C09132=1229.334,-18.388,-40.165,-179.651,5.314,148.817
C09133=1229.329,-18.138,-40.179,-179.649,5.313,148.816
C09134=1229.323,-17.889,-40.193,-179.646,5.314,148.816
C09135=1229.319,-17.639,-40.206,-179.643,5.314,148.815
C09136=1229.314,-17.390,-40.221,-179.641,5.314,148.814
C09137=1229.308,-17.141,-40.235,-179.638,5.315,148.813
C09138=1229.303,-16.890,-40.248,-179.636,5.315,148.813
C09139=1229.299,-16.641,-40.262,-179.634,5.315,148.812
C09140=1229.293,-16.392,-40.276,-179.631,5.315,148.811
C09141=1229.288,-16.142,-40.289,-179.628,5.316,148.810
C09142=1229.283,-15.892,-40.304,-179.626,5.315,148.810
C09143=1229.278,-15.643,-40.317,-179.623,5.316,148.809
C09144=1229.273,-15.394,-40.331,-179.621,5.316,148.808
C09145=1229.268,-15.143,-40.345,-179.618,5.316,148.808
C09146=1229.262,-14.894,-40.359,-179.616,5.316,148.807
C09147=1229.258,-14.645,-40.372,-179.613,5.317,148.806
C09148=1229.253,-14.395,-40.387,-179.611,5.317,148.806
C09149=1229.247,-14.145,-40.400,-179.608,5.317,148.805
C09150=1229.242,-13.896,-40.414,-179.606,5.318,148.804
C09151=1229.237,-13.646,-40.428,-179.604,5.317,148.803
C09152=1229.233,-13.397,-40.442,-179.601,5.318,148.803
C09153=1229.228,-13.148,-40.456,-179.598,5.318,148.802
C09154=1229.222,-12.897,-40.469,-179.596,5.319,148.801
C09155=1229.217,-12.648,-40.483,-179.594,5.319,148.801
C09156=1229.212,-12.399,-40.498,-179.591,5.319,148.800
C09157=1229.208,-12.149,-40.511,-179.588,5.320,148.799
C09158=1229.203,-11.899,-40.526,-179.586,5.319,148.799
C09159=1229.197,-11.650,-40.540,-179.584,5.320,148.798
C09160=1229.192,-11.400,-40.553,-179.581,5.320,148.797
C09161=1229.187,-11.150,-40.567,-179.579,5.320,148.797
C09162=1229.182,-10.901,-40.582,-179.576,5.321,148.796
C09163=1229.176,-10.652,-40.596,-179.573,5.321,148.795
C09164=1229.172,-10.402,-40.609,-179.571,5.321,148.794
C09165=1229.167,-10.153,-40.624,-179.569,5.321,148.794
C09166=1229.162,-9.904,-40.637,-179.566,5.322,148.793
C09167=1229.157,-9.654,-40.652,-179.564,5.322,148.792
C09168=1229.152,-9.404,-40.666,-179.561,5.322,148.792
C09169=1229.147,-9.154,-40.680,-179.559,5.323,148.791
C09170=1229.142,-8.904,-40.694,-179.556,5.323,148.790
C09171=1229.136,-8.655,-40.708,-179.554,5.323,148.790
C09172=1229.131,-8.405,-40.722,-179.551,5.323,148.789
C09173=1229.127,-8.156,-40.736,-179.549,5.324,148.788
C09174=1229.122,-7.906,-40.750,-179.547,5.324,148.788
C09175=1229.116,-7.657,-40.764,-179.544,5.324,148.787
C09176=1229.111,-7.408,-40.778,-179.541,5.325,148.786
C09177=1229.106,-7.158,-40.792,-179.539,5.324,148.785
C09178=1229.102,-6.908,-40.807,-179.537,5.325,148.785
C09179=1229.097,-6.658,-40.821,-179.534,5.325,148.784
C09180=1229.091,-6.409,-40.835,-179.531,5.326,148.783
C09181=1229.086,-6.160,-40.849,-179.529,5.326,148.783
C09182=1229.081,-5.910,-40.863,-179.527,5.326,148.782
C09183=1229.076,-5.660,-40.878,-179.524,5.327,148.781
C09184=1229.071,-5.411,-40.892,-179.522,5.326,148.781
C09185=1229.066,-5.162,-40.906,-179.519,5.327,148.780
C09186=1229.061,-4.912,-40.920,-179.516,5.327,148.779
C09187=1229.056,-4.663,-40.935,-179.514,5.327,148.779
C09188=1229.051,-4.413,-40.949,-179.512,5.328,148.778
C09189=1229.046,-4.163,-40.964,-179.509,5.328,148.777
C09190=1229.041,-3.914,-40.978,-179.506,5.329,148.777
C09191=1229.036,-3.665,-40.992,-179.504,5.328,148.776
C09192=1229.031,-3.415,-41.006,-179.502,5.329,148.775
C09193=1229.026,-3.165,-41.021,-179.499,5.329,148.774
C09194=1229.021,-2.915,-41.035,-179.497,5.329,148.774
C09195=1229.016,-2.666,-41.049,-179.494,5.330,148.773
C09196=1229.011,-2.416,-41.063,-179.492,5.330,148.772
C09197=1229.006,-2.168,-41.078,-179.489,5.331,148.772
C09198=1229.001,-1.918,-41.092,-179.487,5.330,148.771
C09199=1228.996,-1.668,-41.107,-179.484,5.331,148.770
C09200=1228.991,-1.419,-41.121,-179.482,5.331,148.770
C09201=1228.986,-1.169,-41.135,-179.480,5.331,148.769
C09202=1228.981,-0.919,-41.149,-179.477,5.332,148.768
C09203=1228.976,-0.670,-41.164,-179.474,5.332,148.768
C09204=1228.970,-0.420,-41.179,-179.472,5.333,148.767
C09205=1228.965,-0.171,-41.193,-179.469,5.332,148.766
C09206=1228.960,0.079,-41.207,-179.467,5.333,148.765
C09207=1228.955,0.328,-41.222,-179.464,5.334,148.765
C09208=1228.950,0.578,-41.237,-179.462,5.334,148.764
C09209=1228.945,0.827,-41.251,-179.459,5.334,148.763
C09210=1228.940,1.077,-41.265,-179.456,5.334,148.762
C09211=1228.936,1.327,-41.280,-179.454,5.334,148.762
C09212=1228.931,1.576,-41.294,-179.452,5.334,148.761
C09213=1228.925,1.826,-41.309,-179.449,5.335,148.760
C09214=1228.920,2.075,-41.324,-179.446,5.335,148.760
C09215=1228.915,2.324,-41.338,-179.444,5.336,148.759
C09216=1228.910,2.574,-41.353,-179.442,5.335,148.758
C09217=1228.905,2.823,-41.367,-179.439,5.336,148.758
C09218=1228.900,3.073,-41.381,-179.436,5.337,148.757
C09219=1228.894,3.342,-41.397,-179.434,5.337,148.756
C09220=1228.889,3.611,-41.413,-179.431,5.338,148.756
C09221=1228.884,3.880,-41.429,-179.429,5.337,148.755
C09222=1228.879,4.148,-41.445,-179.426,5.338,148.754
C09223=1228.873,4.399,-41.459,-179.424,5.338,148.754
C09224=1228.868,4.648,-41.474,-179.421,5.339,148.753
C09225=1228.864,4.897,-41.489,-179.418,5.339,148.752
C09226=1228.859,5.147,-41.503,-179.416,5.339,148.751
C09227=1228.854,5.396,-41.518,-179.414,5.340,148.751
C09228=1228.848,5.646,-41.533,-179.411,5.340,148.750
C09229=1228.843,5.896,-41.547,-179.408,5.341,148.749
C09230=1228.839,6.145,-41.562,-179.406,5.340,148.749
C09231=1228.834,6.395,-41.576,-179.403,5.341,148.748
C09232=1228.828,6.644,-41.592,-179.401,5.342,148.747
C09233=1228.823,6.894,-41.606,-179.398,5.342,148.747
C09234=1228.818,7.143,-41.621,-179.396,5.342,148.746
C09235=1228.814,7.393,-41.635,-179.393,5.342,148.745
C09236=1228.808,7.643,-41.650,-179.391,5.343,148.745
C09237=1228.803,7.892,-41.665,-179.388,5.343,148.744
C09238=1228.798,8.141,-41.680,-179.386,5.343,148.743
C09239=1228.794,8.390,-41.695,-179.383,5.344,148.743
C09240=1228.788,8.641,-41.710,-179.381,5.344,148.742
C09241=1228.783,8.890,-41.724,-179.378,5.345,148.741
C09242=1228.779,9.139,-41.739,-179.376,5.344,148.740
C09243=1228.773,9.389,-41.754,-179.373,5.345,148.740
C09244=1228.768,9.638,-41.769,-179.371,5.345,148.739
C09245=1228.764,9.888,-41.784,-179.368,5.346,148.738
C09246=1228.759,10.137,-41.798,-179.366,5.346,148.738
C09247=1228.753,10.387,-41.813,-179.363,5.346,148.737
C09248=1228.748,10.636,-41.828,-179.361,5.347,148.736
C09249=1228.744,10.885,-41.843,-179.358,5.347,148.736
C09250=1228.738,11.135,-41.858,-179.356,5.347,148.735
C09251=1228.733,11.385,-41.873,-179.353,5.348,148.734
C09252=1228.728,11.634,-41.888,-179.351,5.348,148.734
C09253=1228.723,11.884,-41.902,-179.348,5.349,148.733
C09254=1228.718,12.133,-41.917,-179.346,5.348,148.732
C09255=1228.713,12.383,-41.932,-179.343,5.349,148.732
C09256=1228.708,12.632,-41.947,-179.341,5.349,148.731
C09257=1228.703,12.882,-41.962,-179.338,5.350,148.730
C09258=1228.698,13.131,-41.977,-179.335,5.351,148.730
C09259=1228.693,13.380,-41.992,-179.333,5.350,148.729
C09260=1228.688,13.631,-42.007,-179.331,5.351,148.728
C09261=1228.683,13.880,-42.022,-179.328,5.351,148.727
C09262=1228.679,14.129,-42.037,-179.325,5.352,148.727
C09263=1228.673,14.379,-42.052,-179.323,5.352,148.726
C09264=1228.668,14.628,-42.067,-179.321,5.352,148.725
C09265=1228.663,14.877,-42.083,-179.318,5.353,148.725
C09266=1228.658,15.127,-42.097,-179.315,5.353,148.724
C09267=1228.653,15.376,-42.112,-179.313,5.354,148.723
C09268=1228.648,15.626,-42.128,-179.311,5.353,148.723
C09269=1228.643,15.875,-42.142,-179.308,5.354,148.722
C09270=1228.638,16.125,-42.158,-179.305,5.355,148.721
C09271=1228.633,16.375,-42.173,-179.303,5.355,148.721
C09272=1228.628,16.624,-42.189,-179.301,5.355,148.720
C09273=1228.623,16.874,-42.203,-179.298,5.355,148.719
C09274=1228.618,17.123,-42.218,-179.295,5.356,148.719
C09275=1228.613,17.372,-42.233,-179.293,5.356,148.718
C09276=1228.608,17.622,-42.249,-179.290,5.357,148.717
C09277=1228.603,17.872,-42.264,-179.288,5.357,148.717
C09278=1228.598,18.121,-42.279,-179.285,5.357,148.716
C09279=1228.593,18.370,-42.294,-179.283,5.358,148.715
C09280=1228.588,18.620,-42.310,-179.280,5.359,148.715
C09281=1228.583,18.869,-42.325,-179.278,5.359,148.714
C09282=1228.578,19.119,-42.340,-179.276,5.359,148.713
C09283=1228.573,19.368,-42.355,-179.273,5.359,148.713
C09284=1228.568,19.618,-42.371,-179.270,5.360,148.712
C09285=1228.563,19.867,-42.386,-179.268,5.361,148.711
C09286=1228.558,20.117,-42.401,-179.265,5.361,148.711
C09287=1228.553,20.366,-42.416,-179.263,5.361,148.710
C09288=1228.548,20.616,-42.431,-179.260,5.361,148.709
C09289=1228.544,20.866,-42.446,-179.258,5.362,148.709
C09290=1228.538,21.115,-42.462,-179.255,5.362,148.708
C09291=1228.533,21.364,-42.478,-179.253,5.363,148.707
C09292=1228.528,21.613,-42.493,-179.250,5.363,148.707
C09293=1228.523,21.863,-42.508,-179.248,5.363,148.706
C09294=1228.519,22.113,-42.524,-179.245,5.364,148.705
C09295=1228.513,22.362,-42.539,-179.243,5.364,148.704
C09296=1228.508,22.612,-42.554,-179.240,5.365,148.704
C09297=1228.503,22.861,-42.569,-179.238,5.365,148.703
C09298=1228.498,23.111,-42.585,-179.235,5.365,148.702
C09299=1228.494,23.360,-42.600,-179.232,5.366,148.702
C09300=1228.488,23.610,-42.616,-179.230,5.366,148.701
C09301=1228.483,23.859,-42.631,-179.227,5.367,148.700
C09302=1228.478,24.108,-42.646,-179.225,5.367,148.700
C09303=1228.473,24.358,-42.662,-179.222,5.367,148.699
C09304=1228.468,24.608,-42.678,-179.220,5.368,148.698
C09305=1228.463,24.857,-42.693,-179.217,5.368,148.698
C09306=1228.458,25.106,-42.708,-179.215,5.369,148.697
C09307=1228.454,25.356,-42.724,-179.212,5.370,148.697
C09308=1228.449,25.605,-42.739,-179.210,5.369,148.696
C09309=1228.443,25.855,-42.755,-179.208,5.370,148.695
C09310=1228.439,26.104,-42.770,-179.205,5.370,148.694
C09311=1228.434,26.354,-42.786,-179.202,5.371,148.694
C09312=1228.428,26.603,-42.801,-179.200,5.372,148.693
C09313=1228.423,26.853,-42.817,-179.197,5.372,148.692
C09314=1228.418,27.102,-42.832,-179.195,5.372,148.692
C09315=1228.414,27.351,-42.849,-179.192,5.372,148.691
C09316=1228.408,27.601,-42.864,-179.190,5.373,148.690
C09317=1228.404,27.850,-42.879,-179.187,5.373,148.690
C09318=1228.399,28.100,-42.895,-179.184,5.374,148.689
C09319=1228.394,28.349,-42.911,-179.182,5.375,148.688
C09320=1228.388,28.599,-42.926,-179.180,5.374,148.688
C09321=1228.384,28.849,-42.942,-179.177,5.375,148.687
C09322=1228.379,29.098,-42.957,-179.174,5.375,148.686
C09323=1228.373,29.367,-42.974,-179.172,5.376,148.686
C09324=1228.368,29.635,-42.991,-179.169,5.377,148.685
C09325=1228.363,29.903,-43.008,-179.167,5.377,148.684
C09326=1228.358,30.172,-43.025,-179.164,5.378,148.684
C09327=1228.353,30.422,-43.041,-179.161,5.378,148.683
C09328=1228.347,30.671,-43.056,-179.159,5.379,148.682
C09329=1228.342,30.921,-43.072,-179.156,5.379,148.682
C09330=1228.338,31.170,-43.087,-179.154,5.379,148.681
C09331=1228.333,31.419,-43.103,-179.151,5.380,148.680
C09332=1228.328,31.669,-43.119,-179.149,5.380,148.680
C09333=1228.322,31.919,-43.135,-179.146,5.381,148.679
C09334=1228.317,32.168,-43.151,-179.143,5.381,148.678
C09335=1228.313,32.417,-43.167,-179.141,5.382,148.678
C09336=1228.308,32.667,-43.182,-179.139,5.382,148.677
C09337=1228.303,32.916,-43.198,-179.136,5.382,148.676
C09338=1228.298,33.166,-43.214,-179.133,5.383,148.675
C09339=1228.293,33.415,-43.230,-179.131,5.383,148.675
C09340=1228.287,33.664,-43.246,-179.129,5.384,148.674
C09341=1228.283,33.914,-43.261,-179.126,5.385,148.674
C09342=1228.278,34.164,-43.277,-179.123,5.385,148.673
C09343=1228.273,34.413,-43.293,-179.121,5.385,148.672
C09344=1228.268,34.662,-43.309,-179.119,5.385,148.672
C09345=1228.263,34.912,-43.324,-179.116,5.386,148.671
C09346=1228.258,35.161,-43.341,-179.113,5.387,148.670
C09347=1228.253,35.411,-43.357,-179.111,5.387,148.670
C09348=1228.248,35.661,-43.373,-179.108,5.388,148.669
C09349=1228.244,35.909,-43.388,-179.105,5.388,148.668
C09350=1228.238,36.159,-43.404,-179.103,5.388,148.668
C09351=1228.233,36.409,-43.420,-179.101,5.389,148.667
C09352=1228.228,36.658,-43.436,-179.098,5.389,148.666
C09353=1228.224,36.908,-43.452,-179.096,5.390,148.666
C09354=1228.219,37.156,-43.469,-179.093,5.391,148.665
C09355=1228.214,37.407,-43.484,-179.091,5.391,148.664
C09356=1228.208,37.656,-43.500,-179.088,5.392,148.664
C09357=1228.203,37.905,-43.516,-179.085,5.392,148.663
C09358=1228.198,38.155,-43.532,-179.083,5.392,148.662
C09359=1228.193,38.404,-43.549,-179.081,5.393,148.662
C09360=1228.189,38.654,-43.565,-179.078,5.393,148.661
C09361=1228.184,38.903,-43.581,-179.075,5.394,148.660
C09362=1228.179,39.153,-43.597,-179.073,5.394,148.660
C09363=1228.173,39.402,-43.612,-179.070,5.395,148.659
C09364=1228.169,39.652,-43.629,-179.067,5.395,148.658
C09365=1228.163,39.901,-43.645,-179.065,5.396,148.658
C09366=1228.159,40.150,-43.661,-179.063,5.396,148.657
C09367=1228.154,40.400,-43.677,-179.060,5.397,148.657
C09368=1228.149,40.649,-43.694,-179.058,5.397,148.656
C09369=1228.144,40.899,-43.709,-179.055,5.398,148.655
C09370=1228.139,41.147,-43.725,-179.053,5.398,148.655
C09371=1228.134,41.398,-43.741,-179.050,5.399,148.654
C09372=1228.129,41.646,-43.758,-179.047,5.399,148.653
C09373=1228.124,41.896,-43.774,-179.045,5.400,148.653
C09374=1228.119,42.145,-43.790,-179.042,5.401,148.652
C09375=1228.114,42.395,-43.807,-179.040,5.400,148.651
C09376=1228.109,42.644,-43.822,-179.038,5.401,148.651
C09377=1228.105,42.894,-43.839,-179.035,5.402,148.650
C09378=1228.100,43.144,-43.855,-179.032,5.402,148.649
C09379=1228.095,43.392,-43.871,-179.030,5.403,148.649
C09380=1228.090,43.642,-43.888,-179.027,5.403,148.648
C09381=1228.085,43.891,-43.903,-179.025,5.404,148.647
C09382=1228.080,44.141,-43.920,-179.022,5.405,148.647
C09383=1228.074,44.391,-43.936,-179.019,5.405,148.646
C09384=1228.070,44.640,-43.953,-179.017,5.406,148.645
C09385=1228.065,44.889,-43.969,-179.015,5.405,148.645
C09386=1228.060,45.139,-43.985,-179.012,5.406,148.644
C09387=1228.055,45.388,-44.002,-179.010,5.407,148.644
C09388=1228.050,45.637,-44.018,-179.007,5.407,148.643
C09389=1228.045,45.887,-44.034,-179.005,5.408,148.642
C09390=1228.040,46.136,-44.050,-179.002,5.409,148.642
C09391=1228.035,46.386,-44.068,-178.999,5.409,148.641
C09392=1228.030,46.635,-44.083,-178.997,5.410,148.640
C09393=1228.025,46.885,-44.100,-178.994,5.410,148.640
C09394=1228.020,47.134,-44.116,-178.991,5.411,148.639
C09395=1228.016,47.383,-44.133,-178.989,5.411,148.638
C09396=1228.010,47.632,-44.149,-178.987,5.412,148.638
C09397=1228.006,47.882,-44.165,-178.984,5.412,148.637
C09398=1228.001,48.132,-44.182,-178.982,5.413,148.636
C09399=1227.996,48.381,-44.199,-178.979,5.413,148.636
C09400=1227.991,48.631,-44.215,-178.977,5.414,148.635
C09401=1227.986,48.879,-44.231,-178.974,5.414,148.634
C09402=1227.981,49.129,-44.248,-178.971,5.415,148.634
C09403=1227.976,49.379,-44.265,-178.969,5.416,148.633
C09404=1227.971,49.627,-44.281,-178.967,5.416,148.633
C09405=1227.966,49.878,-44.297,-178.964,5.417,148.632
C09406=1227.962,50.127,-44.314,-178.961,5.418,148.631
C09407=1227.956,50.376,-44.331,-178.959,5.418,148.631
C09408=1227.951,50.626,-44.347,-178.956,5.419,148.630
C09409=1227.946,50.874,-44.364,-178.954,5.418,148.629
C09410=1227.942,51.124,-44.380,-178.951,5.419,148.629
C09411=1227.936,51.374,-44.397,-178.949,5.420,148.628
C09412=1227.931,51.623,-44.413,-178.946,5.420,148.627
C09413=1227.927,51.873,-44.430,-178.944,5.421,148.627
C09414=1227.922,52.122,-44.447,-178.941,5.422,148.626
C09415=1227.917,52.371,-44.464,-178.939,5.422,148.625
C09416=1227.912,52.621,-44.480,-178.936,5.423,148.625
C09417=1227.908,52.870,-44.497,-178.933,5.423,148.624
C09418=1227.902,53.119,-44.513,-178.931,5.424,148.623
C09419=1227.897,53.369,-44.530,-178.928,5.425,148.623
C09420=1227.892,53.619,-44.546,-178.926,5.425,148.622
C09421=1227.887,53.868,-44.563,-178.923,5.426,148.622
C09422=1227.882,54.117,-44.580,-178.921,5.427,148.621
C09423=1227.878,54.367,-44.597,-178.918,5.427,148.620
C09424=1227.873,54.616,-44.613,-178.915,5.428,148.620
C09425=1227.867,54.865,-44.630,-178.913,5.428,148.619
C09426=1227.863,55.115,-44.647,-178.911,5.428,148.618
C09427=1227.858,55.383,-44.665,-178.907,5.429,148.618
C09428=1227.852,55.652,-44.683,-178.905,5.430,148.617
C09429=1227.847,55.920,-44.701,-178.902,5.431,148.616
C09430=1227.842,56.188,-44.720,-178.900,5.431,148.616
C09431=1227.837,56.438,-44.736,-178.897,5.432,148.615
C09432=1227.832,56.687,-44.753,-178.894,5.432,148.614
C09433=1227.827,56.936,-44.770,-178.892,5.433,148.614
C09434=1227.822,57.186,-44.787,-178.889,5.434,148.613
C09435=1227.817,57.436,-44.804,-178.887,5.434,148.613
C09436=1227.812,57.685,-44.820,-178.884,5.435,148.612
C09437=1227.808,57.934,-44.837,-178.882,5.436,148.611
C09438=1227.802,58.184,-44.854,-178.879,5.436,148.611
C09439=1227.798,58.433,-44.871,-178.876,5.437,148.610
C09440=1227.792,58.682,-44.888,-178.874,5.436,148.609
C09441=1227.788,58.932,-44.904,-178.872,5.437,148.609
C09442=1227.783,59.181,-44.922,-178.869,5.438,148.608
C09443=1227.778,59.431,-44.939,-178.867,5.439,148.607
C09444=1227.772,59.680,-44.956,-178.864,5.439,148.607
C09445=1227.768,59.929,-44.973,-178.862,5.440,148.606
C09446=1227.763,60.179,-44.989,-178.859,5.440,148.605
C09447=1227.758,60.428,-45.006,-178.857,5.441,148.605
C09448=1227.753,60.677,-45.023,-178.854,5.442,148.604
C09449=1227.748,60.926,-45.041,-178.852,5.442,148.604
C09450=1227.744,61.176,-45.057,-178.849,5.443,148.603
C09451=1227.739,61.426,-45.075,-178.846,5.443,148.602
C09452=1227.734,61.675,-45.091,-178.844,5.444,148.602
C09453=1227.728,61.924,-45.108,-178.842,5.445,148.601
C09454=1227.724,62.173,-45.126,-178.839,5.446,148.601
C09455=1227.719,62.423,-45.143,-178.836,5.446,148.600
C09456=1227.714,62.672,-45.160,-178.834,5.447,148.599
C09457=1227.709,62.922,-45.177,-178.831,5.447,148.599
C09458=1227.704,63.170,-45.194,-178.828,5.448,148.598
C09459=1227.699,63.420,-45.211,-178.826,5.448,148.597
C09460=1227.694,63.670,-45.228,-178.824,5.449,148.597
C09461=1227.689,63.919,-45.245,-178.821,5.450,148.596
C09462=1227.685,64.169,-45.263,-178.818,5.451,148.596
C09463=1227.680,64.418,-45.280,-178.816,5.451,148.595
C09464=1227.674,64.667,-45.297,-178.813,5.452,148.594
C09465=1227.670,64.916,-45.314,-178.811,5.453,148.594
C09466=1227.665,65.166,-45.331,-178.808,5.453,148.593
C09467=1227.660,65.416,-45.349,-178.806,5.454,148.592
C09468=1227.655,65.664,-45.366,-178.803,5.454,148.592
C09469=1227.650,65.914,-45.383,-178.800,5.455,148.591
C09470=1227.646,66.164,-45.400,-178.798,5.456,148.590
C09471=1227.641,66.413,-45.418,-178.796,5.457,148.590
C09472=1227.635,66.662,-45.435,-178.793,5.457,148.589
C09473=1227.631,66.911,-45.452,-178.790,5.458,148.589
C09474=1227.626,67.161,-45.469,-178.788,5.458,148.588
C09475=1227.621,67.410,-45.486,-178.785,5.459,148.587
C09476=1227.616,67.659,-45.504,-178.782,5.459,148.587
C09477=1227.611,67.909,-45.521,-178.780,5.460,148.586
C09478=1227.607,68.158,-45.539,-178.778,5.461,148.586
C09479=1227.602,68.408,-45.556,-178.775,5.462,148.585
C09480=1227.596,68.658,-45.573,-178.772,5.462,148.584
C09481=1227.592,68.906,-45.590,-178.770,5.463,148.584
C09482=1227.586,69.156,-45.607,-178.768,5.464,148.583
C09483=1227.582,69.405,-45.625,-178.765,5.464,148.583
C09484=1227.577,69.654,-45.642,-178.762,5.465,148.582
C09485=1227.572,69.903,-45.660,-178.760,5.465,148.581
C09486=1227.567,70.153,-45.677,-178.757,5.466,148.581
C09487=1227.563,70.402,-45.695,-178.755,5.467,148.580
C09488=1227.558,70.652,-45.712,-178.752,5.467,148.579
C09489=1227.553,70.901,-45.730,-178.750,5.468,148.579
C09490=1227.547,71.151,-45.747,-178.747,5.469,148.578
C09491=1227.543,71.400,-45.765,-178.745,5.469,148.577
C09492=1227.538,71.649,-45.783,-178.742,5.470,148.577
C09493=1227.533,71.899,-45.800,-178.740,5.471,148.576
C09494=1227.528,72.148,-45.818,-178.737,5.471,148.576
C09495=1227.524,72.397,-45.835,-178.734,5.472,148.575
C09496=1227.519,72.646,-45.853,-178.731,5.473,148.574
C09497=1227.514,72.896,-45.870,-178.729,5.474,148.574
C09498=1227.509,73.145,-45.888,-178.727,5.475,148.573
C09499=1227.504,73.394,-45.905,-178.724,5.475,148.573
C09500=1227.499,73.643,-45.922,-178.721,5.476,148.572
C09501=1227.494,73.893,-45.940,-178.719,5.477,148.571
C09502=1227.489,74.142,-45.957,-178.717,5.478,148.571
C09503=1227.484,74.392,-45.975,-178.714,5.478,148.570
C09504=1227.479,74.640,-45.993,-178.711,5.479,148.570
C09505=1227.474,74.890,-46.010,-178.709,5.479,148.569
C09506=1227.469,75.139,-46.028,-178.706,5.480,148.568
C09507=1227.464,75.389,-46.046,-178.704,5.481,148.568
C09508=1227.459,75.638,-46.063,-178.701,5.481,148.567
C09509=1227.456,75.888,-46.081,-178.699,5.482,148.567
C09510=1227.451,76.137,-46.099,-178.696,5.483,148.566
C09511=1227.446,76.386,-46.117,-178.694,5.484,148.565
C09512=1227.441,76.636,-46.134,-178.691,5.484,148.565
C09513=1227.436,76.885,-46.152,-178.689,5.485,148.564
C09514=1227.431,77.134,-46.170,-178.686,5.485,148.563
C09515=1227.426,77.384,-46.187,-178.683,5.486,148.563
C09516=1227.421,77.633,-46.205,-178.681,5.487,148.562
C09517=1227.416,77.882,-46.223,-178.678,5.488,148.562
C09518=1227.412,78.131,-46.241,-178.675,5.489,148.561
C09519=1227.407,78.381,-46.259,-178.673,5.490,148.560
C09520=1227.401,78.630,-46.276,-178.671,5.490,148.560
C09521=1227.396,78.880,-46.294,-178.668,5.491,148.559
C09522=1227.392,79.129,-46.312,-178.665,5.492,148.559
C09523=1227.387,79.378,-46.330,-178.663,5.492,148.558
C09524=1227.382,79.627,-46.348,-178.660,5.493,148.557
C09525=1227.377,79.877,-46.365,-178.658,5.494,148.557
C09526=1227.372,80.126,-46.383,-178.655,5.494,148.556
C09527=1227.367,80.375,-46.401,-178.653,5.495,148.556
C09528=1227.362,80.625,-46.419,-178.650,5.496,148.555
C09529=1227.358,80.874,-46.437,-178.648,5.496,148.555
C09530=1227.353,81.123,-46.455,-178.645,5.497,148.554
C09531=1227.347,81.392,-46.474,-178.642,5.498,148.553
C09532=1227.342,81.661,-46.494,-178.640,5.499,148.553
C09533=1227.337,81.929,-46.513,-178.637,5.500,148.552
C09534=1227.332,82.197,-46.532,-178.634,5.500,148.551
C09535=1227.327,82.446,-46.550,-178.632,5.501,148.551
C09536=1227.322,82.695,-46.568,-178.629,5.503,148.550
C09537=1227.317,82.945,-46.586,-178.626,5.503,148.550
C09538=1227.312,83.194,-46.604,-178.624,5.504,148.549
C09539=1227.307,83.443,-46.622,-178.621,5.504,148.548
C09540=1227.302,83.692,-46.640,-178.619,5.505,148.548
C09541=1227.298,83.942,-46.659,-178.616,5.506,148.547
C09542=1227.293,84.192,-46.676,-178.614,5.507,148.547
C09543=1227.288,84.441,-46.694,-178.611,5.507,148.546
C09544=1227.283,84.690,-46.712,-178.609,5.508,148.545
C09545=1227.278,84.939,-46.730,-178.606,5.509,148.545
C09546=1227.274,85.188,-46.748,-178.604,5.509,148.544
C09547=1227.269,85.437,-46.766,-178.601,5.511,148.543
C09548=1227.264,85.687,-46.785,-178.598,5.512,148.543
C09549=1227.259,85.936,-46.803,-178.596,5.512,148.542
C09550=1227.255,86.185,-46.821,-178.593,5.513,148.542
C09551=1227.249,86.435,-46.839,-178.591,5.513,148.541
C09552=1227.244,86.684,-46.857,-178.588,5.514,148.541
C09553=1227.240,86.934,-46.876,-178.586,5.515,148.540
C09554=1227.235,87.183,-46.894,-178.583,5.516,148.539
C09555=1227.230,87.432,-46.912,-178.581,5.516,148.539
C09556=1227.225,87.681,-46.930,-178.578,5.517,148.538
C09557=1227.220,87.931,-46.948,-178.575,5.519,148.538
C09558=1227.216,88.180,-46.966,-178.573,5.519,148.537
C09559=1227.210,88.429,-46.985,-178.570,5.520,148.536
C09560=1227.205,88.678,-47.003,-178.568,5.521,148.536
C09561=1227.201,88.928,-47.021,-178.565,5.521,148.535
C09562=1227.196,89.177,-47.039,-178.563,5.522,148.535
C09563=1227.191,89.427,-47.057,-178.560,5.523,148.534
C09564=1227.186,89.676,-47.075,-178.558,5.523,148.534
C09565=1227.182,89.924,-47.094,-178.555,5.525,148.533
C09566=1227.176,90.174,-47.113,-178.552,5.526,148.532
C09567=1227.172,90.424,-47.131,-178.550,5.526,148.532
C09568=1227.167,90.673,-47.149,-178.547,5.527,148.531
C09569=1227.162,90.922,-47.167,-178.545,5.528,148.531
C09570=1227.157,91.171,-47.186,-178.543,5.529,148.530
C09571=1227.152,91.421,-47.205,-178.540,5.529,148.529
C09572=1227.147,91.670,-47.223,-178.537,5.530,148.529
C09573=1227.143,91.919,-47.241,-178.534,5.531,148.528
C09574=1227.138,92.168,-47.259,-178.532,5.532,148.528
C09575=1227.133,92.418,-47.278,-178.529,5.533,148.527
C09576=1227.128,92.667,-47.296,-178.527,5.533,148.526
C09577=1227.123,92.916,-47.314,-178.525,5.534,148.526
C09578=1227.119,93.166,-47.333,-178.522,5.535,148.525
C09579=1227.113,93.415,-47.352,-178.519,5.536,148.525
C09580=1227.108,93.664,-47.370,-178.517,5.536,148.524
C09581=1227.104,93.913,-47.389,-178.514,5.538,148.524
C09582=1227.100,94.163,-47.407,-178.511,5.539,148.523
C09583=1227.094,94.412,-47.425,-178.509,5.539,148.522
C09584=1227.089,94.661,-47.444,-178.507,5.540,148.522
C09585=1227.085,94.911,-47.462,-178.504,5.541,148.521
C09586=1227.079,95.160,-47.481,-178.501,5.541,148.521
C09587=1227.075,95.409,-47.500,-178.499,5.543,148.520
C09588=1227.070,95.659,-47.518,-178.496,5.544,148.520
C09589=1227.065,95.907,-47.537,-178.494,5.544,148.519
C09590=1227.060,96.157,-47.555,-178.491,5.545,148.518
C09591=1227.056,96.406,-47.574,-178.489,5.546,148.518
C09592=1227.051,96.655,-47.593,-178.486,5.546,148.517
C09593=1227.046,96.904,-47.611,-178.484,5.547,148.517
C09594=1227.042,97.154,-47.630,-178.481,5.549,148.516
C09595=1227.036,97.403,-47.649,-178.478,5.549,148.515
C09596=1227.031,97.652,-47.667,-178.476,5.550,148.515
C09597=1227.027,97.902,-47.686,-178.473,5.551,148.514
C09598=1227.022,98.151,-47.705,-178.471,5.552,148.514
C09599=1227.017,98.400,-47.723,-178.468,5.552,148.513
C09600=1227.012,98.649,-47.743,-178.466,5.554,148.513
C09601=1227.007,98.898,-47.761,-178.463,5.555,148.512
C09602=1227.003,99.148,-47.780,-178.460,5.555,148.511
C09603=1226.997,99.397,-47.798,-178.458,5.556,148.511
C09604=1226.993,99.646,-47.817,-178.456,5.557,148.510
C09605=1226.988,99.896,-47.836,-178.453,5.557,148.510
C09606=1226.983,100.144,-47.855,-178.450,5.559,148.509
C09607=1226.978,100.395,-47.873,-178.448,5.560,148.509
C09608=1226.974,100.643,-47.892,-178.445,5.560,148.508
C09609=1226.969,100.892,-47.910,-178.443,5.561,148.508
C09610=1226.964,101.142,-47.930,-178.440,5.562,148.507
C09611=1226.959,101.391,-47.949,-178.437,5.563,148.506
C09612=1226.954,101.641,-47.967,-178.435,5.564,148.506
C09613=1226.950,101.889,-47.986,-178.432,5.565,148.505
C09614=1226.945,102.139,-48.005,-178.430,5.566,148.505
C09615=1226.940,102.388,-48.024,-178.428,5.567,148.504
C09616=1226.935,102.637,-48.043,-178.425,5.567,148.504
C09617=1226.930,102.887,-48.061,-178.422,5.569,148.503
C09618=1226.925,103.136,-48.081,-178.420,5.570,148.502
C09619=1226.921,103.385,-48.100,-178.417,5.570,148.502
C09620=1226.915,103.634,-48.118,-178.414,5.571,148.501
C09621=1226.911,103.884,-48.137,-178.412,5.572,148.501
C09622=1226.906,104.133,-48.157,-178.409,5.573,148.500
C09623=1226.902,104.382,-48.175,-178.407,5.574,148.499
C09624=1226.896,104.631,-48.194,-178.404,5.575,148.499
C09625=1226.892,104.881,-48.213,-178.402,5.575,148.498
C09626=1226.887,105.129,-48.233,-178.399,5.576,148.498
C09627=1226.881,105.379,-48.251,-178.397,5.578,148.497
C09628=1226.877,105.628,-48.270,-178.394,5.578,148.497
C09629=1226.872,105.877,-48.290,-178.391,5.579,148.496
C09630=1226.868,106.126,-48.309,-178.389,5.580,148.496
C09631=1226.862,106.376,-48.327,-178.387,5.581,148.495
C09632=1226.858,106.625,-48.346,-178.383,5.582,148.494
C09633=1226.853,106.874,-48.366,-178.381,5.583,148.494
C09634=1226.848,107.123,-48.385,-178.379,5.584,148.493
C09635=1226.843,107.392,-48.405,-178.376,5.584,148.493
C09636=1226.838,107.660,-48.426,-178.373,5.586,148.492
C09637=1226.833,107.929,-48.447,-178.371,5.587,148.492
C09638=1226.828,108.197,-48.468,-178.368,5.588,148.491
C09639=1226.823,108.447,-48.487,-178.365,5.589,148.490
C09640=1226.818,108.696,-48.505,-178.363,5.590,148.490
C09641=1226.813,108.945,-48.525,-178.360,5.590,148.489
C09642=1226.808,109.194,-48.544,-178.357,5.592,148.489
C09643=1226.804,109.443,-48.563,-178.355,5.593,148.488
C09644=1226.799,109.692,-48.582,-178.352,5.593,148.488
C09645=1226.794,109.942,-48.602,-178.350,5.594,148.487
C09646=1226.789,110.190,-48.621,-178.348,5.595,148.487
C09647=1226.785,110.440,-48.641,-178.344,5.596,148.486
C09648=1226.780,110.689,-48.660,-178.342,5.597,148.486
C09649=1226.775,110.939,-48.678,-178.340,5.598,148.485
C09650=1226.770,111.188,-48.698,-178.337,5.599,148.484
C09651=1226.765,111.437,-48.717,-178.334,5.600,148.484
C09652=1226.760,111.687,-48.737,-178.332,5.601,148.483
C09653=1226.756,111.935,-48.755,-178.329,5.602,148.483
C09654=1226.751,112.185,-48.775,-178.327,5.603,148.482
C09655=1226.746,112.434,-48.795,-178.324,5.604,148.482
C09656=1226.741,112.683,-48.813,-178.322,5.605,148.481
C09657=1226.737,112.932,-48.833,-178.319,5.606,148.480
C09658=1226.731,113.181,-48.852,-178.316,5.606,148.480
C09659=1226.727,113.431,-48.872,-178.314,5.608,148.479
C09660=1226.723,113.680,-48.891,-178.311,5.609,148.479
C09661=1226.717,113.929,-48.910,-178.309,5.610,148.478
C09662=1226.713,114.178,-48.931,-178.306,5.610,148.478
C09663=1226.707,114.427,-48.950,-178.303,5.612,148.477
C09664=1226.703,114.676,-48.970,-178.301,5.613,148.477
C09665=1226.699,114.926,-48.989,-178.299,5.613,148.476
C09666=1226.693,115.175,-49.008,-178.296,5.614,148.476
C09667=1226.689,115.424,-49.028,-178.293,5.616,148.475
C09668=1226.684,115.674,-49.047,-178.291,5.616,148.474
C09669=1226.679,115.923,-49.067,-178.288,5.617,148.474
C09670=1226.674,116.172,-49.086,-178.286,5.618,148.473
C09671=1226.670,116.421,-49.105,-178.283,5.620,148.473
C09672=1226.665,116.670,-49.125,-178.281,5.620,148.472
C09673=1226.660,116.919,-49.145,-178.278,5.621,148.472
C09674=1226.655,117.169,-49.165,-178.276,5.622,148.471
C09675=1226.650,117.418,-49.184,-178.273,5.623,148.471
C09676=1226.645,117.667,-49.204,-178.271,5.624,148.470
C09677=1226.641,117.916,-49.224,-178.268,5.625,148.470
C09678=1226.636,118.165,-49.243,-178.265,5.627,148.469
C09679=1226.631,118.414,-49.262,-178.263,5.627,148.469
C09680=1226.627,118.664,-49.282,-178.260,5.628,148.468
C09681=1226.621,118.913,-49.301,-178.258,5.629,148.467
C09682=1226.617,119.162,-49.322,-178.255,5.630,148.467
C09683=1226.612,119.411,-49.341,-178.253,5.631,148.466
C09684=1226.607,119.661,-49.361,-178.250,5.632,148.466
C09685=1226.602,119.910,-49.380,-178.247,5.633,148.465
C09686=1226.598,120.159,-49.401,-178.245,5.634,148.465
C09687=1226.593,120.408,-49.420,-178.242,5.635,148.464
C09688=1226.588,120.657,-49.440,-178.240,5.636,148.464
C09689=1226.583,120.906,-49.460,-178.237,5.637,148.463
C09690=1226.578,121.156,-49.480,-178.235,5.638,148.463
C09691=1226.574,121.405,-49.499,-178.232,5.639,148.462
C09692=1226.569,121.653,-49.519,-178.229,5.640,148.461
C09693=1226.564,121.903,-49.539,-178.227,5.641,148.461
C09694=1226.560,122.152,-49.558,-178.224,5.642,148.460
C09695=1226.555,122.401,-49.578,-178.222,5.643,148.460
C09696=1226.550,122.650,-49.598,-178.219,5.644,148.459
C09697=1226.545,122.900,-49.617,-178.217,5.645,148.459
C09698=1226.541,123.149,-49.638,-178.214,5.646,148.458
C09699=1226.535,123.398,-49.658,-178.212,5.648,148.458
C09700=1226.530,123.647,-49.678,-178.209,5.649,148.457
C09701=1226.526,123.896,-49.698,-178.206,5.649,148.457
C09702=1226.521,124.146,-49.717,-178.204,5.651,148.456
C09703=1226.516,124.395,-49.738,-178.201,5.652,148.456
C09704=1226.512,124.644,-49.757,-178.199,5.653,148.455
C09705=1226.507,124.893,-49.777,-178.196,5.654,148.455
C09706=1226.502,125.142,-49.797,-178.194,5.655,148.454
C09707=1226.497,125.391,-49.817,-178.191,5.656,148.454
C09708=1226.493,125.641,-49.837,-178.189,5.657,148.453
C09709=1226.488,125.890,-49.857,-178.186,5.658,148.453
C09710=1226.483,126.138,-49.877,-178.184,5.659,148.452
C09711=1226.478,126.387,-49.897,-178.181,5.660,148.452
C09712=1226.474,126.637,-49.917,-178.178,5.661,148.451
C09713=1226.469,126.886,-49.937,-178.176,5.662,148.450
C09714=1226.465,127.136,-49.957,-178.173,5.663,148.450
C09715=1226.459,127.385,-49.978,-178.170,5.664,148.449
C09716=1226.454,127.634,-49.997,-178.168,5.665,148.449
C09717=1226.450,127.883,-50.017,-178.166,5.666,148.448
C09718=1226.445,128.132,-50.038,-178.163,5.668,148.448
C09719=1226.440,128.381,-50.057,-178.160,5.669,148.447
C09720=1226.436,128.630,-50.078,-178.158,5.669,148.447
C09721=1226.431,128.880,-50.097,-178.155,5.671,148.446
C09722=1226.426,129.129,-50.118,-178.153,5.672,148.446
C09723=1226.421,129.377,-50.138,-178.150,5.673,148.445
C09724=1226.416,129.627,-50.158,-178.147,5.674,148.445
C09725=1226.412,129.876,-50.178,-178.145,5.675,148.444
C09726=1226.407,130.125,-50.199,-178.143,5.676,148.444
C09727=1226.403,130.374,-50.218,-178.140,5.677,148.443
C09728=1226.398,130.623,-50.239,-178.137,5.678,148.443
C09729=1226.393,130.872,-50.260,-178.135,5.679,148.442
C09730=1226.388,131.122,-50.279,-178.132,5.681,148.442
C09731=1226.384,131.371,-50.300,-178.130,5.681,148.441
C09732=1226.378,131.619,-50.320,-178.127,5.683,148.441
C09733=1226.373,131.869,-50.340,-178.125,5.684,148.440
C09734=1226.369,132.118,-50.360,-178.122,5.685,148.440
C09735=1226.364,132.367,-50.381,-178.119,5.686,148.439
C09736=1226.359,132.616,-50.402,-178.117,5.687,148.439
C09737=1226.355,132.866,-50.421,-178.114,5.688,148.438
C09738=1226.350,133.115,-50.442,-178.111,5.689,148.438
C09739=1226.345,133.383,-50.464,-178.109,5.690,148.437
C09740=1226.340,133.652,-50.485,-178.106,5.692,148.437
C09741=1226.335,133.921,-50.508,-178.104,5.693,148.436
C09742=1226.329,134.190,-50.530,-178.100,5.694,148.435
C09743=1226.325,134.439,-50.550,-178.098,5.695,148.435
C09744=1226.321,134.688,-50.570,-178.095,5.696,148.434
C09745=1226.315,134.937,-50.591,-178.093,5.697,148.434
C09746=1226.311,135.186,-50.612,-178.090,5.698,148.433
C09747=1226.307,135.435,-50.632,-178.088,5.700,148.433
C09748=1226.301,135.685,-50.652,-178.085,5.700,148.432
C09749=1226.297,135.934,-50.673,-178.083,5.702,148.432
C09750=1226.292,136.182,-50.693,-178.080,5.703,148.431
C09751=1226.286,136.431,-50.714,-178.078,5.704,148.431
C09752=1226.282,136.680,-50.734,-178.075,5.705,148.430
C09753=1226.277,136.929,-50.755,-178.073,5.706,148.430
C09754=1226.272,137.178,-50.775,-178.070,5.707,148.429
C09755=1226.268,137.427,-50.796,-178.067,5.709,148.429
C09756=1226.263,137.676,-50.817,-178.065,5.709,148.428
C09757=1226.258,137.925,-50.837,-178.062,5.711,148.428
C09758=1226.254,138.174,-50.858,-178.059,5.712,148.427
C09759=1226.249,138.424,-50.879,-178.057,5.713,148.427
C09760=1226.245,138.673,-50.899,-178.055,5.715,148.426
C09761=1226.240,138.923,-50.920,-178.052,5.715,148.426
C09762=1226.235,139.171,-50.941,-178.049,5.717,148.425
C09763=1226.230,139.421,-50.962,-178.047,5.718,148.425
C09764=1226.226,139.670,-50.982,-178.045,5.719,148.424
C09765=1226.221,139.919,-51.002,-178.041,5.720,148.424
C09766=1226.216,140.168,-51.023,-178.039,5.721,148.423
C09767=1226.212,140.417,-51.044,-178.036,5.723,148.423
C09768=1226.206,140.666,-51.065,-178.034,5.724,148.422
C09769=1226.202,140.915,-51.085,-178.031,5.724,148.422
C09770=1226.197,141.164,-51.106,-178.029,5.726,148.421
C09771=1226.192,141.413,-51.126,-178.026,5.727,148.421
C09772=1226.187,141.663,-51.147,-178.024,5.729,148.420
C09773=1226.183,141.911,-51.168,-178.021,5.730,148.420
C09774=1226.178,142.161,-51.189,-178.019,5.730,148.419
C09775=1226.173,142.410,-51.209,-178.016,5.732,148.419
C09776=1226.168,142.658,-51.231,-178.014,5.733,148.418
C09777=1226.164,142.908,-51.251,-178.011,5.734,148.418
C09778=1226.159,143.157,-51.272,-178.008,5.735,148.417
C09779=1226.155,143.406,-51.293,-178.006,5.737,148.417
C09780=1226.150,143.655,-51.314,-178.003,5.738,148.416
C09781=1226.145,143.904,-51.334,-178.001,5.739,148.416
C09782=1226.140,144.153,-51.356,-177.998,5.740,148.415
C09783=1226.135,144.402,-51.377,-177.996,5.741,148.415
C09784=1226.131,144.651,-51.397,-177.993,5.743,148.414
C09785=1226.126,144.900,-51.418,-177.990,5.743,148.414
C09786=1226.122,145.150,-51.439,-177.988,5.745,148.413
C09787=1226.117,145.399,-51.461,-177.985,5.746,148.413
C09788=1226.112,145.648,-51.481,-177.983,5.747,148.412
C09789=1226.107,145.897,-51.502,-177.980,5.748,148.412
C09790=1226.102,146.146,-51.523,-177.978,5.749,148.411
C09791=1226.098,146.395,-51.544,-177.975,5.751,148.411
C09792=1226.093,146.644,-51.565,-177.972,5.752,148.410
C09793=1226.089,146.893,-51.586,-177.970,5.754,148.410
C09794=1226.084,147.142,-51.607,-177.967,5.754,148.409
C09795=1226.079,147.391,-51.628,-177.965,5.756,148.409
C09796=1226.074,147.640,-51.649,-177.962,5.757,148.408
C09797=1226.070,147.889,-51.670,-177.960,5.758,148.408
C09798=1226.064,148.138,-51.691,-177.957,5.760,148.408
C09799=1226.061,148.388,-51.712,-177.955,5.760,148.407
C09800=1226.056,148.637,-51.734,-177.952,5.762,148.407
C09801=1226.051,148.886,-51.755,-177.949,5.763,148.406
C09802=1226.046,149.135,-51.775,-177.947,5.764,148.406
C09803=1226.041,149.383,-51.797,-177.945,5.765,148.405
C09804=1226.037,149.633,-51.818,-177.941,5.767,148.405
C09805=1226.032,149.882,-51.840,-177.939,5.768,148.404
C09806=1226.027,150.131,-51.860,-177.936,5.769,148.404
C09807=1226.022,150.380,-51.881,-177.934,5.770,148.403
C09808=1226.017,150.629,-51.903,-177.932,5.771,148.403
C09809=1226.013,150.878,-51.924,-177.929,5.773,148.402
C09810=1226.009,151.127,-51.945,-177.927,5.774,148.402
C09811=1226.003,151.376,-51.966,-177.924,5.775,148.401
C09812=1225.999,151.625,-51.988,-177.921,5.776,148.401
C09813=1225.995,151.875,-52.009,-177.919,5.778,148.401
C09814=1225.990,152.123,-52.030,-177.916,5.779,148.400
C09815=1225.985,152.373,-52.051,-177.914,5.781,148.400
C09816=1225.980,152.621,-52.073,-177.911,5.781,148.399
C09817=1225.975,152.871,-52.094,-177.908,5.783,148.399
C09818=1225.971,153.119,-52.115,-177.906,5.784,148.398
C09819=1225.966,153.369,-52.136,-177.903,5.786,148.398
C09820=1225.961,153.617,-52.158,-177.901,5.787,148.397
C09821=1225.956,153.867,-52.179,-177.898,5.788,148.397
C09822=1225.952,154.116,-52.201,-177.896,5.789,148.396
C09823=1225.947,154.364,-52.222,-177.893,5.791,148.396
C09824=1225.942,154.614,-52.243,-177.890,5.791,148.395
C09825=1225.938,154.863,-52.265,-177.888,5.793,148.395
C09826=1225.933,155.112,-52.286,-177.886,5.794,148.394
C09827=1225.928,155.361,-52.308,-177.882,5.796,148.394
C09828=1225.924,155.610,-52.330,-177.880,5.797,148.393
C09829=1225.919,155.859,-52.351,-177.877,5.798,148.393
C09830=1225.914,156.108,-52.372,-177.875,5.799,148.392
C09831=1225.910,156.357,-52.394,-177.872,5.801,148.392
C09832=1225.905,156.606,-52.415,-177.870,5.802,148.391
C09833=1225.900,156.855,-52.437,-177.867,5.804,148.391
C09834=1225.896,157.104,-52.459,-177.865,5.805,148.391
C09835=1225.891,157.354,-52.480,-177.862,5.806,148.390
C09836=1225.886,157.602,-52.501,-177.860,5.807,148.390
C09837=1225.882,157.852,-52.523,-177.857,5.809,148.389
C09838=1225.877,158.100,-52.545,-177.855,5.809,148.389
C09839=1225.871,158.349,-52.566,-177.852,5.811,148.388
C09840=1225.868,158.598,-52.587,-177.849,5.812,148.388
C09841=1225.863,158.847,-52.609,-177.847,5.814,148.387
C09842=1225.858,159.096,-52.631,-177.845,5.815,148.387
C09843=1225.853,159.365,-52.654,-177.841,5.816,148.386
C09844=1225.847,159.634,-52.677,-177.839,5.818,148.386
C09845=1225.843,159.904,-52.701,-177.836,5.819,148.385
C09846=1225.838,160.173,-52.725,-177.834,5.821,148.385
C09847=1225.833,160.422,-52.746,-177.830,5.822,148.384
C09848=1225.828,160.670,-52.768,-177.828,5.823,148.384
C09849=1225.824,160.920,-52.790,-177.826,5.825,148.384
C09850=1225.819,161.169,-52.811,-177.823,5.826,148.383
C09851=1225.814,161.418,-52.833,-177.820,5.827,148.383
C09852=1225.810,161.667,-52.855,-177.818,5.828,148.382
C09853=1225.805,161.915,-52.876,-177.815,5.830,148.382
C09854=1225.800,162.165,-52.899,-177.813,5.831,148.381
C09855=1225.796,162.413,-52.920,-177.810,5.833,148.381
C09856=1225.791,162.663,-52.942,-177.808,5.833,148.380
C09857=1225.786,162.911,-52.964,-177.805,5.835,148.380
C09858=1225.782,163.160,-52.986,-177.802,5.837,148.380
C09859=1225.777,163.409,-53.008,-177.800,5.838,148.379
C09860=1225.772,163.659,-53.029,-177.797,5.839,148.379
C09861=1225.768,163.908,-53.051,-177.795,5.840,148.378
C09862=1225.763,164.157,-53.072,-177.792,5.842,148.378
C09863=1225.758,164.406,-53.095,-177.790,5.843,148.377
C09864=1225.753,164.655,-53.117,-177.787,5.845,148.377
C09865=1225.749,164.904,-53.139,-177.785,5.845,148.376
C09866=1225.744,165.153,-53.160,-177.782,5.847,148.376
C09867=1225.740,165.402,-53.182,-177.779,5.849,148.376
C09868=1225.735,165.651,-53.204,-177.777,5.850,148.375
C09869=1225.731,165.900,-53.227,-177.774,5.852,148.375
C09870=1225.726,166.148,-53.249,-177.772,5.853,148.374
C09871=1225.720,166.397,-53.271,-177.769,5.854,148.374
C09872=1225.716,166.647,-53.293,-177.767,5.855,148.373
C09873=1225.711,166.895,-53.315,-177.764,5.857,148.373
C09874=1225.707,167.145,-53.337,-177.762,5.858,148.372
C09875=1225.702,167.393,-53.358,-177.759,5.859,148.372
C09876=1225.698,167.643,-53.380,-177.756,5.861,148.371
C09877=1225.692,167.891,-53.403,-177.754,5.862,148.371
C09878=1225.688,168.141,-53.425,-177.751,5.864,148.370
C09879=1225.684,168.390,-53.447,-177.749,5.865,148.370
C09880=1225.679,168.638,-53.469,-177.746,5.866,148.370
C09881=1225.675,168.888,-53.491,-177.743,5.868,148.369
C09882=1225.669,169.136,-53.513,-177.741,5.869,148.369
C09883=1225.665,169.386,-53.536,-177.738,5.871,148.368
C09884=1225.660,169.634,-53.557,-177.736,5.872,148.368
C09885=1225.656,169.883,-53.580,-177.733,5.873,148.367
C09886=1225.651,170.132,-53.602,-177.731,5.874,148.367
C09887=1225.646,170.381,-53.624,-177.728,5.876,148.367
C09888=1225.641,170.630,-53.646,-177.725,5.878,148.366
C09889=1225.637,170.879,-53.668,-177.723,5.879,148.366
C09890=1225.632,171.128,-53.691,-177.720,5.880,148.365
C09891=1225.628,171.377,-53.713,-177.718,5.881,148.365
C09892=1225.623,171.626,-53.735,-177.715,5.883,148.364
C09893=1225.618,171.875,-53.758,-177.712,5.885,148.364
C09894=1225.614,172.124,-53.780,-177.710,5.886,148.364
C09895=1225.609,172.373,-53.802,-177.707,5.887,148.363
C09896=1225.605,172.622,-53.824,-177.705,5.888,148.363
C09897=1225.600,172.871,-53.847,-177.702,5.890,148.362
C09898=1225.595,173.120,-53.869,-177.700,5.892,148.362
C09899=1225.591,173.369,-53.891,-177.697,5.893,148.361
C09900=1225.586,173.617,-53.914,-177.695,5.894,148.361
C09901=1225.581,173.867,-53.936,-177.693,5.895,148.361
C09902=1225.577,174.116,-53.959,-177.690,5.897,148.360
C09903=1225.572,174.364,-53.981,-177.687,5.899,148.360
C09904=1225.567,174.614,-54.003,-177.685,5.900,148.359
C09905=1225.562,174.862,-54.026,-177.682,5.902,148.359
C09906=1225.558,175.112,-54.048,-177.679,5.903,148.359
C09907=1225.554,175.360,-54.071,-177.677,5.904,148.358
C09908=1225.548,175.609,-54.093,-177.674,5.906,148.358
C09909=1225.544,175.859,-54.115,-177.672,5.907,148.357
C09910=1225.539,176.108,-54.139,-177.669,5.909,148.357
C09911=1225.534,176.356,-54.160,-177.666,5.910,148.356
C09912=1225.530,176.605,-54.184,-177.664,5.911,148.356
C09913=1225.525,176.855,-54.206,-177.661,5.913,148.356
C09914=1225.521,177.103,-54.228,-177.659,5.915,148.355
C09915=1225.516,177.352,-54.251,-177.656,5.916,148.355
C09916=1225.512,177.601,-54.274,-177.654,5.917,148.354
C09917=1225.506,177.850,-54.296,-177.651,5.918,148.354
C09918=1225.502,178.099,-54.319,-177.649,5.920,148.353
C09919=1225.497,178.348,-54.341,-177.646,5.922,148.353
C09920=1225.493,178.596,-54.364,-177.644,5.923,148.352
C09921=1225.488,178.845,-54.387,-177.641,5.925,148.352
C09922=1225.484,179.095,-54.409,-177.638,5.926,148.352
C09923=1225.479,179.344,-54.432,-177.636,5.927,148.351
C09924=1225.474,179.592,-54.454,-177.633,5.929,148.351
C09925=1225.470,179.841,-54.477,-177.630,5.931,148.350
C09926=1225.466,180.090,-54.500,-177.628,5.932,148.350
C09927=1225.460,180.339,-54.522,-177.626,5.934,148.350
C09928=1225.456,180.588,-54.545,-177.623,5.935,148.349
C09929=1225.451,180.837,-54.568,-177.620,5.936,148.349
C09930=1225.447,181.086,-54.591,-177.618,5.938,148.348
C09931=1225.442,181.334,-54.614,-177.615,5.940,148.348
C09932=1225.437,181.584,-54.636,-177.613,5.941,148.347
C09933=1225.433,181.833,-54.659,-177.610,5.942,148.347
C09934=1225.428,182.082,-54.682,-177.607,5.944,148.347
C09935=1225.424,182.330,-54.705,-177.605,5.945,148.346
C09936=1225.419,182.580,-54.727,-177.603,5.947,148.346
C09937=1225.415,182.828,-54.750,-177.599,5.949,148.345
C09938=1225.410,183.077,-54.774,-177.597,5.950,148.345
C09939=1225.405,183.326,-54.797,-177.595,5.951,148.345
C09940=1225.400,183.575,-54.819,-177.592,5.953,148.344
C09941=1225.396,183.824,-54.842,-177.590,5.954,148.344
C09942=1225.392,184.073,-54.865,-177.587,5.956,148.343
C09943=1225.387,184.322,-54.888,-177.584,5.958,148.343
C09944=1225.381,184.571,-54.910,-177.582,5.959,148.343
C09945=1225.377,184.819,-54.933,-177.579,5.960,148.342
C09946=1225.373,185.068,-54.956,-177.577,5.962,148.342
C09947=1225.367,185.338,-54.981,-177.574,5.964,148.341
C09948=1225.363,185.608,-55.006,-177.572,5.965,148.341
C09949=1225.357,185.877,-55.031,-177.568,5.966,148.340
C09950=1225.352,186.147,-55.056,-177.566,5.968,148.340
C09951=1225.348,186.396,-55.079,-177.563,5.970,148.340
C09952=1225.343,186.645,-55.102,-177.560,5.972,148.339
C09953=1225.339,186.894,-55.125,-177.558,5.972,148.339
C09954=1225.335,187.143,-55.148,-177.555,5.974,148.338
C09955=1225.330,187.391,-55.171,-177.553,5.976,148.338
C09956=1225.325,187.640,-55.195,-177.551,5.977,148.338
C09957=1225.320,187.889,-55.218,-177.548,5.979,148.337
C09958=1225.316,188.138,-55.241,-177.545,5.981,148.337
C09959=1225.311,188.387,-55.264,-177.542,5.982,148.336
C09960=1225.307,188.636,-55.287,-177.540,5.983,148.336
C09961=1225.302,188.885,-55.311,-177.537,5.985,148.336
C09962=1225.297,189.133,-55.333,-177.535,5.987,148.335
C09963=1225.293,189.382,-55.357,-177.533,5.988,148.335
C09964=1225.288,189.631,-55.380,-177.530,5.990,148.335
C09965=1225.283,189.880,-55.403,-177.527,5.991,148.334
C09966=1225.279,190.129,-55.427,-177.524,5.993,148.334
C09967=1225.275,190.378,-55.449,-177.522,5.994,148.333
C09968=1225.270,190.627,-55.473,-177.519,5.996,148.333
C09969=1225.265,190.876,-55.496,-177.517,5.998,148.333
C09970=1225.261,191.125,-55.519,-177.515,5.999,148.332
C09971=1225.256,191.374,-55.543,-177.512,6.000,148.332
C09972=1225.251,191.622,-55.566,-177.509,6.002,148.331
C09973=1225.247,191.871,-55.589,-177.506,6.004,148.331
C09974=1225.242,192.120,-55.612,-177.504,6.005,148.331
C09975=1225.237,192.369,-55.635,-177.502,6.007,148.330
C09976=1225.233,192.617,-55.659,-177.499,6.009,148.330
C09977=1225.228,192.867,-55.683,-177.496,6.011,148.330
C09978=1225.223,193.116,-55.706,-177.494,6.011,148.329
C09979=1225.219,193.365,-55.729,-177.491,6.013,148.329
C09980=1225.214,193.614,-55.753,-177.488,6.015,148.328
C09981=1225.209,193.863,-55.776,-177.486,6.016,148.328
C09982=1225.206,194.111,-55.800,-177.484,6.018,148.328
C09983=1225.201,194.360,-55.823,-177.481,6.020,148.327
C09984=1225.196,194.609,-55.846,-177.478,6.022,148.327
C09985=1225.192,194.858,-55.870,-177.476,6.022,148.326
C09986=1225.187,195.107,-55.893,-177.473,6.024,148.326
C09987=1225.183,195.355,-55.917,-177.471,6.026,148.326
C09988=1225.178,195.604,-55.941,-177.468,6.028,148.325
C09989=1225.173,195.853,-55.964,-177.466,6.029,148.325
C09990=1225.168,196.102,-55.987,-177.463,6.031,148.324
C09991=1225.164,196.351,-56.011,-177.461,6.033,148.324
C09992=1225.159,196.600,-56.035,-177.458,6.034,148.324
C09993=1225.155,196.849,-56.058,-177.455,6.036,148.323
C09994=1225.150,197.097,-56.082,-177.453,6.037,148.323
C09995=1225.146,197.346,-56.105,-177.450,6.039,148.323
C09996=1225.141,197.595,-56.129,-177.447,6.041,148.322
//INST
///DATE 2021/06/25 14:26
///ATTR SC,RW,RJ
////FRAME ROBOT
///GROUP1 RB1
NOP
MOVL C00000 V=800.0 PL=0
MOVL C00001 V=800.0 PL=0
MOVL C00002 V=800.0 PL=0
MOVL C00003 V=800.0 PL=0
MOVL C00004 V=800.0 PL=0
MOVL C00005 V=800.0 PL=0
MOVL C00006 V=800.0 PL=0
MOVL C00007 V=800.0 PL=0
MOVL C00008 V=800.0 PL=0
MOVL C00009 V=800.0 PL=0
MOVL C00010 V=800.0 PL=0
MOVL C00011 V=800.0 PL=0
MOVL C00012 V=800.0 PL=0
MOVL C00013 V=800.0 PL=0
MOVL C00014 V=800.0 PL=0
MOVL C00015 V=800.0 PL=0
MOVL C00016 V=800.0 PL=0
MOVL C00017 V=800.0 PL=0
MOVL C00018 V=800.0 PL=0
MOVL C00019 V=800.0 PL=0
MOVL C00020 V=800.0 PL=0
MOVL C00021 V=800.0 PL=0
MOVL C00022 V=800.0 PL=0
MOVL C00023 V=800.0 PL=0
MOVL C00024 V=800.0 PL=0
MOVL C00025 V=800.0 PL=0
MOVL C00026 V=800.0 PL=0
MOVL C00027 V=800.0 PL=0
MOVL C00028 V=800.0 PL=0
MOVL C00029 V=800.0 PL=0
MOVL C00030 V=800.0 PL=0
MOVL C00031 V=800.0 PL=0
MOVL C00032 V=800.0 PL=0
MOVL C00033 V=800.0 PL=0
MOVL C00034 V=800.0 PL=0
MOVL C00035 V=800.0 PL=0
MOVL C00036 V=800.0 PL=0
MOVL C00037 V=800.0 PL=0
MOVL C00038 V=800.0 PL=0
MOVL C00039 V=800.0 PL=0
MOVL C00040 V=800.0 PL=0
MOVL C00041 V=800.0 PL=0
MOVL C00042 V=800.0 PL=0
MOVL C00043 V=800.0 PL=0
MOVL C00044 V=800.0 PL=0
MOVL C00045 V=800.0 PL=0
MOVL C00046 V=800.0 PL=0
MOVL C00047 V=800.0 PL=0
MOVL C00048 V=800.0 PL=0
MOVL C00049 V=800.0 PL=0
MOVL C00050 V=800.0 PL=0
MOVL C00051 V=800.0 PL=0
MOVL C00052 V=800.0 PL=0
MOVL C00053 V=800.0 PL=0
MOVL C00054 V=800.0 PL=0
MOVL C00055 V=800.0 PL=0
MOVL C00056 V=800.0 PL=0
MOVL C00057 V=800.0 PL=0
MOVL C00058 V=800.0 PL=0
MOVL C00059 V=800.0 PL=0
MOVL C00060 V=800.0 PL=0
MOVL C00061 V=800.0 PL=0
MOVL C00062 V=800.0 PL=0
MOVL C00063 V=800.0 PL=0
MOVL C00064 V=800.0 PL=0
MOVL C00065 V=800.0 PL=0
MOVL C00066 V=800.0 PL=0
MOVL C00067 V=800.0 PL=0
MOVL C00068 V=800.0 PL=0
MOVL C00069 V=800.0 PL=0
MOVL C00070 V=800.0 PL=0
MOVL C00071 V=800.0 PL=0
MOVL C00072 V=800.0 PL=0
MOVL C00073 V=800.0 PL=0
MOVL C00074 V=800.0 PL=0
MOVL C00075 V=800.0 PL=0
MOVL C00076 V=800.0 PL=0
MOVL C00077 V=800.0 PL=0
MOVL C00078 V=800.0 PL=0
MOVL C00079 V=800.0 PL=0
MOVL C00080 V=800.0 PL=0
MOVL C00081 V=800.0 PL=0
MOVL C00082 V=800.0 PL=0
MOVL C00083 V=800.0 PL=0
MOVL C00084 V=800.0 PL=0
MOVL C00085 V=800.0 PL=0
MOVL C00086 V=800.0 PL=0
MOVL C00087 V=800.0 PL=0
MOVL C00088 V=800.0 PL=0
MOVL C00089 V=800.0 PL=0
MOVL C00090 V=800.0 PL=0
MOVL C00091 V=800.0 PL=0
MOVL C00092 V=800.0 PL=0
MOVL C00093 V=800.0 PL=0
MOVL C00094 V=800.0 PL=0
MOVL C00095 V=800.0 PL=0
MOVL C00096 V=800.0 PL=0
MOVL C00097 V=800.0 PL=0
MOVL C00098 V=800.0 PL=0
MOVL C00099 V=800.0 PL=0
MOVL C00100 V=800.0 PL=0
MOVL C00101 V=800.0 PL=0
MOVL C00102 V=800.0 PL=0
MOVL C00103 V=800.0 PL=0
MOVL C00104 V=800.0 PL=0
MOVL C00105 V=800.0 PL=0
MOVL C00106 V=800.0 PL=0
MOVL C00107 V=800.0 PL=0
MOVL C00108 V=800.0 PL=0
MOVL C00109 V=800.0 PL=0
MOVL C00110 V=800.0 PL=0
MOVL C00111 V=800.0 PL=0
MOVL C00112 V=800.0 PL=0
MOVL C00113 V=800.0 PL=0
MOVL C00114 V=800.0 PL=0
MOVL C00115 V=800.0 PL=0
MOVL C00116 V=800.0 PL=0
MOVL C00117 V=800.0 PL=0
MOVL C00118 V=800.0 PL=0
MOVL C00119 V=800.0 PL=0
MOVL C00120 V=800.0 PL=0
MOVL C00121 V=800.0 PL=0
MOVL C00122 V=800.0 PL=0
MOVL C00123 V=800.0 PL=0
MOVL C00124 V=800.0 PL=0
MOVL C00125 V=800.0 PL=0
MOVL C00126 V=800.0 PL=0
MOVL C00127 V=800.0 PL=0
MOVL C00128 V=800.0 PL=0
MOVL C00129 V=800.0 PL=0
MOVL C00130 V=800.0 PL=0
MOVL C00131 V=800.0 PL=0
MOVL C00132 V=800.0 PL=0
MOVL C00133 V=800.0 PL=0
MOVL C00134 V=800.0 PL=0
MOVL C00135 V=800.0 PL=0
MOVL C00136 V=800.0 PL=0
MOVL C00137 V=800.0 PL=0
MOVL C00138 V=800.0 PL=0
MOVL C00139 V=800.0 PL=0
MOVL C00140 V=800.0 PL=0
MOVL C00141 V=800.0 PL=0
MOVL C00142 V=800.0 PL=0
MOVL C00143 V=800.0 PL=0
MOVL C00144 V=800.0 PL=0
MOVL C00145 V=800.0 PL=0
MOVL C00146 V=800.0 PL=0
MOVL C00147 V=800.0 PL=0
MOVL C00148 V=800.0 PL=0
MOVL C00149 V=800.0 PL=0
MOVL C00150 V=800.0 PL=0
MOVL C00151 V=800.0 PL=0
MOVL C00152 V=800.0 PL=0
MOVL C00153 V=800.0 PL=0
MOVL C00154 V=800.0 PL=0
MOVL C00155 V=800.0 PL=0
MOVL C00156 V=800.0 PL=0
MOVL C00157 V=800.0 PL=0
MOVL C00158 V=800.0 PL=0
MOVL C00159 V=800.0 PL=0
MOVL C00160 V=800.0 PL=0
MOVL C00161 V=800.0 PL=0
MOVL C00162 V=800.0 PL=0
MOVL C00163 V=800.0 PL=0
MOVL C00164 V=800.0 PL=0
MOVL C00165 V=800.0 PL=0
MOVL C00166 V=800.0 PL=0
MOVL C00167 V=800.0 PL=0
MOVL C00168 V=800.0 PL=0
MOVL C00169 V=800.0 PL=0
MOVL C00170 V=800.0 PL=0
MOVL C00171 V=800.0 PL=0
MOVL C00172 V=800.0 PL=0
MOVL C00173 V=800.0 PL=0
MOVL C00174 V=800.0 PL=0
MOVL C00175 V=800.0 PL=0
MOVL C00176 V=800.0 PL=0
MOVL C00177 V=800.0 PL=0
MOVL C00178 V=800.0 PL=0
MOVL C00179 V=800.0 PL=0
MOVL C00180 V=800.0 PL=0
MOVL C00181 V=800.0 PL=0
MOVL C00182 V=800.0 PL=0
MOVL C00183 V=800.0 PL=0
MOVL C00184 V=800.0 PL=0
MOVL C00185 V=800.0 PL=0
MOVL C00186 V=800.0 PL=0
MOVL C00187 V=800.0 PL=0
MOVL C00188 V=800.0 PL=0
MOVL C00189 V=800.0 PL=0
MOVL C00190 V=800.0 PL=0
MOVL C00191 V=800.0 PL=0
MOVL C00192 V=800.0 PL=0
MOVL C00193 V=800.0 PL=0
MOVL C00194 V=800.0 PL=0
MOVL C00195 V=800.0 PL=0
MOVL C00196 V=800.0 PL=0
MOVL C00197 V=800.0 PL=0
MOVL C00198 V=800.0 PL=0
MOVL C00199 V=800.0 PL=0
MOVL C00200 V=800.0 PL=0
MOVL C00201 V=800.0 PL=0
MOVL C00202 V=800.0 PL=0
MOVL C00203 V=800.0 PL=0
MOVL C00204 V=800.0 PL=0
MOVL C00205 V=800.0 PL=0
MOVL C00206 V=800.0 PL=0
MOVL C00207 V=800.0 PL=0
MOVL C00208 V=800.0 PL=0
MOVL C00209 V=800.0 PL=0
MOVL C00210 V=800.0 PL=0
MOVL C00211 V=800.0 PL=0
MOVL C00212 V=800.0 PL=0
MOVL C00213 V=800.0 PL=0
MOVL C00214 V=800.0 PL=0
MOVL C00215 V=800.0 PL=0
MOVL C00216 V=800.0 PL=0
MOVL C00217 V=800.0 PL=0
MOVL C00218 V=800.0 PL=0
MOVL C00219 V=800.0 PL=0
MOVL C00220 V=800.0 PL=0
MOVL C00221 V=800.0 PL=0
MOVL C00222 V=800.0 PL=0
MOVL C00223 V=800.0 PL=0
MOVL C00224 V=800.0 PL=0
MOVL C00225 V=800.0 PL=0
MOVL C00226 V=800.0 PL=0
MOVL C00227 V=800.0 PL=0
MOVL C00228 V=800.0 PL=0
MOVL C00229 V=800.0 PL=0
MOVL C00230 V=800.0 PL=0
MOVL C00231 V=800.0 PL=0
MOVL C00232 V=800.0 PL=0
MOVL C00233 V=800.0 PL=0
MOVL C00234 V=800.0 PL=0
MOVL C00235 V=800.0 PL=0
MOVL C00236 V=800.0 PL=0
MOVL C00237 V=800.0 PL=0
MOVL C00238 V=800.0 PL=0
MOVL C00239 V=800.0 PL=0
MOVL C00240 V=800.0 PL=0
MOVL C00241 V=800.0 PL=0
MOVL C00242 V=800.0 PL=0
MOVL C00243 V=800.0 PL=0
MOVL C00244 V=800.0 PL=0
MOVL C00245 V=800.0 PL=0
MOVL C00246 V=800.0 PL=0
MOVL C00247 V=800.0 PL=0
MOVL C00248 V=800.0 PL=0
MOVL C00249 V=800.0 PL=0
MOVL C00250 V=800.0 PL=0
MOVL C00251 V=800.0 PL=0
MOVL C00252 V=800.0 PL=0
MOVL C00253 V=800.0 PL=0
MOVL C00254 V=800.0 PL=0
MOVL C00255 V=800.0 PL=0
MOVL C00256 V=800.0 PL=0
MOVL C00257 V=800.0 PL=0
MOVL C00258 V=800.0 PL=0
MOVL C00259 V=800.0 PL=0
MOVL C00260 V=800.0 PL=0
MOVL C00261 V=800.0 PL=0
MOVL C00262 V=800.0 PL=0
MOVL C00263 V=800.0 PL=0
MOVL C00264 V=800.0 PL=0
MOVL C00265 V=800.0 PL=0
MOVL C00266 V=800.0 PL=0
MOVL C00267 V=800.0 PL=0
MOVL C00268 V=800.0 PL=0
MOVL C00269 V=800.0 PL=0
MOVL C00270 V=800.0 PL=0
MOVL C00271 V=800.0 PL=0
MOVL C00272 V=800.0 PL=0
MOVL C00273 V=800.0 PL=0
MOVL C00274 V=800.0 PL=0
MOVL C00275 V=800.0 PL=0
MOVL C00276 V=800.0 PL=0
MOVL C00277 V=800.0 PL=0
MOVL C00278 V=800.0 PL=0
MOVL C00279 V=800.0 PL=0
MOVL C00280 V=800.0 PL=0
MOVL C00281 V=800.0 PL=0
MOVL C00282 V=800.0 PL=0
MOVL C00283 V=800.0 PL=0
MOVL C00284 V=800.0 PL=0
MOVL C00285 V=800.0 PL=0
MOVL C00286 V=800.0 PL=0
MOVL C00287 V=800.0 PL=0
MOVL C00288 V=800.0 PL=0
MOVL C00289 V=800.0 PL=0
MOVL C00290 V=800.0 PL=0
MOVL C00291 V=800.0 PL=0
MOVL C00292 V=800.0 PL=0
MOVL C00293 V=800.0 PL=0
MOVL C00294 V=800.0 PL=0
MOVL C00295 V=800.0 PL=0
MOVL C00296 V=800.0 PL=0
MOVL C00297 V=800.0 PL=0
MOVL C00298 V=800.0 PL=0
MOVL C00299 V=800.0 PL=0
MOVL C00300 V=800.0 PL=0
MOVL C00301 V=800.0 PL=0
MOVL C00302 V=800.0 PL=0
MOVL C00303 V=800.0 PL=0
MOVL C00304 V=800.0 PL=0
MOVL C00305 V=800.0 PL=0
MOVL C00306 V=800.0 PL=0
MOVL C00307 V=800.0 PL=0
MOVL C00308 V=800.0 PL=0
MOVL C00309 V=800.0 PL=0
MOVL C00310 V=800.0 PL=0
MOVL C00311 V=800.0 PL=0
MOVL C00312 V=800.0 PL=0
MOVL C00313 V=800.0 PL=0
MOVL C00314 V=800.0 PL=0
MOVL C00315 V=800.0 PL=0
MOVL C00316 V=800.0 PL=0
MOVL C00317 V=800.0 PL=0
MOVL C00318 V=800.0 PL=0
MOVL C00319 V=800.0 PL=0
MOVL C00320 V=800.0 PL=0
MOVL C00321 V=800.0 PL=0
MOVL C00322 V=800.0 PL=0
MOVL C00323 V=800.0 PL=0
MOVL C00324 V=800.0 PL=0
MOVL C00325 V=800.0 PL=0
MOVL C00326 V=800.0 PL=0
MOVL C00327 V=800.0 PL=0
MOVL C00328 V=800.0 PL=0
MOVL C00329 V=800.0 PL=0
MOVL C00330 V=800.0 PL=0
MOVL C00331 V=800.0 PL=0
MOVL C00332 V=800.0 PL=0
MOVL C00333 V=800.0 PL=0
MOVL C00334 V=800.0 PL=0
MOVL C00335 V=800.0 PL=0
MOVL C00336 V=800.0 PL=0
MOVL C00337 V=800.0 PL=0
MOVL C00338 V=800.0 PL=0
MOVL C00339 V=800.0 PL=0
MOVL C00340 V=800.0 PL=0
MOVL C00341 V=800.0 PL=0
MOVL C00342 V=800.0 PL=0
MOVL C00343 V=800.0 PL=0
MOVL C00344 V=800.0 PL=0
MOVL C00345 V=800.0 PL=0
MOVL C00346 V=800.0 PL=0
MOVL C00347 V=800.0 PL=0
MOVL C00348 V=800.0 PL=0
MOVL C00349 V=800.0 PL=0
MOVL C00350 V=800.0 PL=0
MOVL C00351 V=800.0 PL=0
MOVL C00352 V=800.0 PL=0
MOVL C00353 V=800.0 PL=0
MOVL C00354 V=800.0 PL=0
MOVL C00355 V=800.0 PL=0
MOVL C00356 V=800.0 PL=0
MOVL C00357 V=800.0 PL=0
MOVL C00358 V=800.0 PL=0
MOVL C00359 V=800.0 PL=0
MOVL C00360 V=800.0 PL=0
MOVL C00361 V=800.0 PL=0
MOVL C00362 V=800.0 PL=0
MOVL C00363 V=800.0 PL=0
MOVL C00364 V=800.0 PL=0
MOVL C00365 V=800.0 PL=0
MOVL C00366 V=800.0 PL=0
MOVL C00367 V=800.0 PL=0
MOVL C00368 V=800.0 PL=0
MOVL C00369 V=800.0 PL=0
MOVL C00370 V=800.0 PL=0
MOVL C00371 V=800.0 PL=0
MOVL C00372 V=800.0 PL=0
MOVL C00373 V=800.0 PL=0
MOVL C00374 V=800.0 PL=0
MOVL C00375 V=800.0 PL=0
MOVL C00376 V=800.0 PL=0
MOVL C00377 V=800.0 PL=0
MOVL C00378 V=800.0 PL=0
MOVL C00379 V=800.0 PL=0
MOVL C00380 V=800.0 PL=0
MOVL C00381 V=800.0 PL=0
MOVL C00382 V=800.0 PL=0
MOVL C00383 V=800.0 PL=0
MOVL C00384 V=800.0 PL=0
MOVL C00385 V=800.0 PL=0
MOVL C00386 V=800.0 PL=0
MOVL C00387 V=800.0 PL=0
MOVL C00388 V=800.0 PL=0
MOVL C00389 V=800.0 PL=0
MOVL C00390 V=800.0 PL=0
MOVL C00391 V=800.0 PL=0
MOVL C00392 V=800.0 PL=0
MOVL C00393 V=800.0 PL=0
MOVL C00394 V=800.0 PL=0
MOVL C00395 V=800.0 PL=0
MOVL C00396 V=800.0 PL=0
MOVL C00397 V=800.0 PL=0
MOVL C00398 V=800.0 PL=0
MOVL C00399 V=800.0 PL=0
MOVL C00400 V=800.0 PL=0
MOVL C00401 V=800.0 PL=0
MOVL C00402 V=800.0 PL=0
MOVL C00403 V=800.0 PL=0
MOVL C00404 V=800.0 PL=0
MOVL C00405 V=800.0 PL=0
MOVL C00406 V=800.0 PL=0
MOVL C00407 V=800.0 PL=0
MOVL C00408 V=800.0 PL=0
MOVL C00409 V=800.0 PL=0
MOVL C00410 V=800.0 PL=0
MOVL C00411 V=800.0 PL=0
MOVL C00412 V=800.0 PL=0
MOVL C00413 V=800.0 PL=0
MOVL C00414 V=800.0 PL=0
MOVL C00415 V=800.0 PL=0
MOVL C00416 V=800.0 PL=0
MOVL C00417 V=800.0 PL=0
MOVL C00418 V=800.0 PL=0
MOVL C00419 V=800.0 PL=0
MOVL C00420 V=800.0 PL=0
MOVL C00421 V=800.0 PL=0
MOVL C00422 V=800.0 PL=0
MOVL C00423 V=800.0 PL=0
MOVL C00424 V=800.0 PL=0
MOVL C00425 V=800.0 PL=0
MOVL C00426 V=800.0 PL=0
MOVL C00427 V=800.0 PL=0
MOVL C00428 V=800.0 PL=0
MOVL C00429 V=800.0 PL=0
MOVL C00430 V=800.0 PL=0
MOVL C00431 V=800.0 PL=0
MOVL C00432 V=800.0 PL=0
MOVL C00433 V=800.0 PL=0
MOVL C00434 V=800.0 PL=0
MOVL C00435 V=800.0 PL=0
MOVL C00436 V=800.0 PL=0
MOVL C00437 V=800.0 PL=0
MOVL C00438 V=800.0 PL=0
MOVL C00439 V=800.0 PL=0
MOVL C00440 V=800.0 PL=0
MOVL C00441 V=800.0 PL=0
MOVL C00442 V=800.0 PL=0
MOVL C00443 V=800.0 PL=0
MOVL C00444 V=800.0 PL=0
MOVL C00445 V=800.0 PL=0
MOVL C00446 V=800.0 PL=0
MOVL C00447 V=800.0 PL=0
MOVL C00448 V=800.0 PL=0
MOVL C00449 V=800.0 PL=0
MOVL C00450 V=800.0 PL=0
MOVL C00451 V=800.0 PL=0
MOVL C00452 V=800.0 PL=0
MOVL C00453 V=800.0 PL=0
MOVL C00454 V=800.0 PL=0
MOVL C00455 V=800.0 PL=0
MOVL C00456 V=800.0 PL=0
MOVL C00457 V=800.0 PL=0
MOVL C00458 V=800.0 PL=0
MOVL C00459 V=800.0 PL=0
MOVL C00460 V=800.0 PL=0
MOVL C00461 V=800.0 PL=0
MOVL C00462 V=800.0 PL=0
MOVL C00463 V=800.0 PL=0
MOVL C00464 V=800.0 PL=0
MOVL C00465 V=800.0 PL=0
MOVL C00466 V=800.0 PL=0
MOVL C00467 V=800.0 PL=0
MOVL C00468 V=800.0 PL=0
MOVL C00469 V=800.0 PL=0
MOVL C00470 V=800.0 PL=0
MOVL C00471 V=800.0 PL=0
MOVL C00472 V=800.0 PL=0
MOVL C00473 V=800.0 PL=0
MOVL C00474 V=800.0 PL=0
MOVL C00475 V=800.0 PL=0
MOVL C00476 V=800.0 PL=0
MOVL C00477 V=800.0 PL=0
MOVL C00478 V=800.0 PL=0
MOVL C00479 V=800.0 PL=0
MOVL C00480 V=800.0 PL=0
MOVL C00481 V=800.0 PL=0
MOVL C00482 V=800.0 PL=0
MOVL C00483 V=800.0 PL=0
MOVL C00484 V=800.0 PL=0
MOVL C00485 V=800.0 PL=0
MOVL C00486 V=800.0 PL=0
MOVL C00487 V=800.0 PL=0
MOVL C00488 V=800.0 PL=0
MOVL C00489 V=800.0 PL=0
MOVL C00490 V=800.0 PL=0
MOVL C00491 V=800.0 PL=0
MOVL C00492 V=800.0 PL=0
MOVL C00493 V=800.0 PL=0
MOVL C00494 V=800.0 PL=0
MOVL C00495 V=800.0 PL=0
MOVL C00496 V=800.0 PL=0
MOVL C00497 V=800.0 PL=0
MOVL C00498 V=800.0 PL=0
MOVL C00499 V=800.0 PL=0
MOVL C00500 V=800.0 PL=0
MOVL C00501 V=800.0 PL=0
MOVL C00502 V=800.0 PL=0
MOVL C00503 V=800.0 PL=0
MOVL C00504 V=800.0 PL=0
MOVL C00505 V=800.0 PL=0
MOVL C00506 V=800.0 PL=0
MOVL C00507 V=800.0 PL=0
MOVL C00508 V=800.0 PL=0
MOVL C00509 V=800.0 PL=0
MOVL C00510 V=800.0 PL=0
MOVL C00511 V=800.0 PL=0
MOVL C00512 V=800.0 PL=0
MOVL C00513 V=800.0 PL=0
MOVL C00514 V=800.0 PL=0
MOVL C00515 V=800.0 PL=0
MOVL C00516 V=800.0 PL=0
MOVL C00517 V=800.0 PL=0
MOVL C00518 V=800.0 PL=0
MOVL C00519 V=800.0 PL=0
MOVL C00520 V=800.0 PL=0
MOVL C00521 V=800.0 PL=0
MOVL C00522 V=800.0 PL=0
MOVL C00523 V=800.0 PL=0
MOVL C00524 V=800.0 PL=0
MOVL C00525 V=800.0 PL=0
MOVL C00526 V=800.0 PL=0
MOVL C00527 V=800.0 PL=0
MOVL C00528 V=800.0 PL=0
MOVL C00529 V=800.0 PL=0
MOVL C00530 V=800.0 PL=0
MOVL C00531 V=800.0 PL=0
MOVL C00532 V=800.0 PL=0
MOVL C00533 V=800.0 PL=0
MOVL C00534 V=800.0 PL=0
MOVL C00535 V=800.0 PL=0
MOVL C00536 V=800.0 PL=0
MOVL C00537 V=800.0 PL=0
MOVL C00538 V=800.0 PL=0
MOVL C00539 V=800.0 PL=0
MOVL C00540 V=800.0 PL=0
MOVL C00541 V=800.0 PL=0
MOVL C00542 V=800.0 PL=0
MOVL C00543 V=800.0 PL=0
MOVL C00544 V=800.0 PL=0
MOVL C00545 V=800.0 PL=0
MOVL C00546 V=800.0 PL=0
MOVL C00547 V=800.0 PL=0
MOVL C00548 V=800.0 PL=0
MOVL C00549 V=800.0 PL=0
MOVL C00550 V=800.0 PL=0
MOVL C00551 V=800.0 PL=0
MOVL C00552 V=800.0 PL=0
MOVL C00553 V=800.0 PL=0
MOVL C00554 V=800.0 PL=0
MOVL C00555 V=800.0 PL=0
MOVL C00556 V=800.0 PL=0
MOVL C00557 V=800.0 PL=0
MOVL C00558 V=800.0 PL=0
MOVL C00559 V=800.0 PL=0
MOVL C00560 V=800.0 PL=0
MOVL C00561 V=800.0 PL=0
MOVL C00562 V=800.0 PL=0
MOVL C00563 V=800.0 PL=0
MOVL C00564 V=800.0 PL=0
MOVL C00565 V=800.0 PL=0
MOVL C00566 V=800.0 PL=0
MOVL C00567 V=800.0 PL=0
MOVL C00568 V=800.0 PL=0
MOVL C00569 V=800.0 PL=0
MOVL C00570 V=800.0 PL=0
MOVL C00571 V=800.0 PL=0
MOVL C00572 V=800.0 PL=0
MOVL C00573 V=800.0 PL=0
MOVL C00574 V=800.0 PL=0
MOVL C00575 V=800.0 PL=0
MOVL C00576 V=800.0 PL=0
MOVL C00577 V=800.0 PL=0
MOVL C00578 V=800.0 PL=0
MOVL C00579 V=800.0 PL=0
MOVL C00580 V=800.0 PL=0
MOVL C00581 V=800.0 PL=0
MOVL C00582 V=800.0 PL=0
MOVL C00583 V=800.0 PL=0
MOVL C00584 V=800.0 PL=0
MOVL C00585 V=800.0 PL=0
MOVL C00586 V=800.0 PL=0
MOVL C00587 V=800.0 PL=0
MOVL C00588 V=800.0 PL=0
MOVL C00589 V=800.0 PL=0
MOVL C00590 V=800.0 PL=0
MOVL C00591 V=800.0 PL=0
MOVL C00592 V=800.0 PL=0
MOVL C00593 V=800.0 PL=0
MOVL C00594 V=800.0 PL=0
MOVL C00595 V=800.0 PL=0
MOVL C00596 V=800.0 PL=0
MOVL C00597 V=800.0 PL=0
MOVL C00598 V=800.0 PL=0
MOVL C00599 V=800.0 PL=0
MOVL C00600 V=800.0 PL=0
MOVL C00601 V=800.0 PL=0
MOVL C00602 V=800.0 PL=0
MOVL C00603 V=800.0 PL=0
MOVL C00604 V=800.0 PL=0
MOVL C00605 V=800.0 PL=0
MOVL C00606 V=800.0 PL=0
MOVL C00607 V=800.0 PL=0
MOVL C00608 V=800.0 PL=0
MOVL C00609 V=800.0 PL=0
MOVL C00610 V=800.0 PL=0
MOVL C00611 V=800.0 PL=0
MOVL C00612 V=800.0 PL=0
MOVL C00613 V=800.0 PL=0
MOVL C00614 V=800.0 PL=0
MOVL C00615 V=800.0 PL=0
MOVL C00616 V=800.0 PL=0
MOVL C00617 V=800.0 PL=0
MOVL C00618 V=800.0 PL=0
MOVL C00619 V=800.0 PL=0
MOVL C00620 V=800.0 PL=0
MOVL C00621 V=800.0 PL=0
MOVL C00622 V=800.0 PL=0
MOVL C00623 V=800.0 PL=0
MOVL C00624 V=800.0 PL=0
MOVL C00625 V=800.0 PL=0
MOVL C00626 V=800.0 PL=0
MOVL C00627 V=800.0 PL=0
MOVL C00628 V=800.0 PL=0
MOVL C00629 V=800.0 PL=0
MOVL C00630 V=800.0 PL=0
MOVL C00631 V=800.0 PL=0
MOVL C00632 V=800.0 PL=0
MOVL C00633 V=800.0 PL=0
MOVL C00634 V=800.0 PL=0
MOVL C00635 V=800.0 PL=0
MOVL C00636 V=800.0 PL=0
MOVL C00637 V=800.0 PL=0
MOVL C00638 V=800.0 PL=0
MOVL C00639 V=800.0 PL=0
MOVL C00640 V=800.0 PL=0
MOVL C00641 V=800.0 PL=0
MOVL C00642 V=800.0 PL=0
MOVL C00643 V=800.0 PL=0
MOVL C00644 V=800.0 PL=0
MOVL C00645 V=800.0 PL=0
MOVL C00646 V=800.0 PL=0
MOVL C00647 V=800.0 PL=0
MOVL C00648 V=800.0 PL=0
MOVL C00649 V=800.0 PL=0
MOVL C00650 V=800.0 PL=0
MOVL C00651 V=800.0 PL=0
MOVL C00652 V=800.0 PL=0
MOVL C00653 V=800.0 PL=0
MOVL C00654 V=800.0 PL=0
MOVL C00655 V=800.0 PL=0
MOVL C00656 V=800.0 PL=0
MOVL C00657 V=800.0 PL=0
MOVL C00658 V=800.0 PL=0
MOVL C00659 V=800.0 PL=0
MOVL C00660 V=800.0 PL=0
MOVL C00661 V=800.0 PL=0
MOVL C00662 V=800.0 PL=0
MOVL C00663 V=800.0 PL=0
MOVL C00664 V=800.0 PL=0
MOVL C00665 V=800.0 PL=0
MOVL C00666 V=800.0 PL=0
MOVL C00667 V=800.0 PL=0
MOVL C00668 V=800.0 PL=0
MOVL C00669 V=800.0 PL=0
MOVL C00670 V=800.0 PL=0
MOVL C00671 V=800.0 PL=0
MOVL C00672 V=800.0 PL=0
MOVL C00673 V=800.0 PL=0
MOVL C00674 V=800.0 PL=0
MOVL C00675 V=800.0 PL=0
MOVL C00676 V=800.0 PL=0
MOVL C00677 V=800.0 PL=0
MOVL C00678 V=800.0 PL=0
MOVL C00679 V=800.0 PL=0
MOVL C00680 V=800.0 PL=0
MOVL C00681 V=800.0 PL=0
MOVL C00682 V=800.0 PL=0
MOVL C00683 V=800.0 PL=0
MOVL C00684 V=800.0 PL=0
MOVL C00685 V=800.0 PL=0
MOVL C00686 V=800.0 PL=0
MOVL C00687 V=800.0 PL=0
MOVL C00688 V=800.0 PL=0
MOVL C00689 V=800.0 PL=0
MOVL C00690 V=800.0 PL=0
MOVL C00691 V=800.0 PL=0
MOVL C00692 V=800.0 PL=0
MOVL C00693 V=800.0 PL=0
MOVL C00694 V=800.0 PL=0
MOVL C00695 V=800.0 PL=0
MOVL C00696 V=800.0 PL=0
MOVL C00697 V=800.0 PL=0
MOVL C00698 V=800.0 PL=0
MOVL C00699 V=800.0 PL=0
MOVL C00700 V=800.0 PL=0
MOVL C00701 V=800.0 PL=0
MOVL C00702 V=800.0 PL=0
MOVL C00703 V=800.0 PL=0
MOVL C00704 V=800.0 PL=0
MOVL C00705 V=800.0 PL=0
MOVL C00706 V=800.0 PL=0
MOVL C00707 V=800.0 PL=0
MOVL C00708 V=800.0 PL=0
MOVL C00709 V=800.0 PL=0
MOVL C00710 V=800.0 PL=0
MOVL C00711 V=800.0 PL=0
MOVL C00712 V=800.0 PL=0
MOVL C00713 V=800.0 PL=0
MOVL C00714 V=800.0 PL=0
MOVL C00715 V=800.0 PL=0
MOVL C00716 V=800.0 PL=0
MOVL C00717 V=800.0 PL=0
MOVL C00718 V=800.0 PL=0
MOVL C00719 V=800.0 PL=0
MOVL C00720 V=800.0 PL=0
MOVL C00721 V=800.0 PL=0
MOVL C00722 V=800.0 PL=0
MOVL C00723 V=800.0 PL=0
MOVL C00724 V=800.0 PL=0
MOVL C00725 V=800.0 PL=0
MOVL C00726 V=800.0 PL=0
MOVL C00727 V=800.0 PL=0
MOVL C00728 V=800.0 PL=0
MOVL C00729 V=800.0 PL=0
MOVL C00730 V=800.0 PL=0
MOVL C00731 V=800.0 PL=0
MOVL C00732 V=800.0 PL=0
MOVL C00733 V=800.0 PL=0
MOVL C00734 V=800.0 PL=0
MOVL C00735 V=800.0 PL=0
MOVL C00736 V=800.0 PL=0
MOVL C00737 V=800.0 PL=0
MOVL C00738 V=800.0 PL=0
MOVL C00739 V=800.0 PL=0
MOVL C00740 V=800.0 PL=0
MOVL C00741 V=800.0 PL=0
MOVL C00742 V=800.0 PL=0
MOVL C00743 V=800.0 PL=0
MOVL C00744 V=800.0 PL=0
MOVL C00745 V=800.0 PL=0
MOVL C00746 V=800.0 PL=0
MOVL C00747 V=800.0 PL=0
MOVL C00748 V=800.0 PL=0
MOVL C00749 V=800.0 PL=0
MOVL C00750 V=800.0 PL=0
MOVL C00751 V=800.0 PL=0
MOVL C00752 V=800.0 PL=0
MOVL C00753 V=800.0 PL=0
MOVL C00754 V=800.0 PL=0
MOVL C00755 V=800.0 PL=0
MOVL C00756 V=800.0 PL=0
MOVL C00757 V=800.0 PL=0
MOVL C00758 V=800.0 PL=0
MOVL C00759 V=800.0 PL=0
MOVL C00760 V=800.0 PL=0
MOVL C00761 V=800.0 PL=0
MOVL C00762 V=800.0 PL=0
MOVL C00763 V=800.0 PL=0
MOVL C00764 V=800.0 PL=0
MOVL C00765 V=800.0 PL=0
MOVL C00766 V=800.0 PL=0
MOVL C00767 V=800.0 PL=0
MOVL C00768 V=800.0 PL=0
MOVL C00769 V=800.0 PL=0
MOVL C00770 V=800.0 PL=0
MOVL C00771 V=800.0 PL=0
MOVL C00772 V=800.0 PL=0
MOVL C00773 V=800.0 PL=0
MOVL C00774 V=800.0 PL=0
MOVL C00775 V=800.0 PL=0
MOVL C00776 V=800.0 PL=0
MOVL C00777 V=800.0 PL=0
MOVL C00778 V=800.0 PL=0
MOVL C00779 V=800.0 PL=0
MOVL C00780 V=800.0 PL=0
MOVL C00781 V=800.0 PL=0
MOVL C00782 V=800.0 PL=0
MOVL C00783 V=800.0 PL=0
MOVL C00784 V=800.0 PL=0
MOVL C00785 V=800.0 PL=0
MOVL C00786 V=800.0 PL=0
MOVL C00787 V=800.0 PL=0
MOVL C00788 V=800.0 PL=0
MOVL C00789 V=800.0 PL=0
MOVL C00790 V=800.0 PL=0
MOVL C00791 V=800.0 PL=0
MOVL C00792 V=800.0 PL=0
MOVL C00793 V=800.0 PL=0
MOVL C00794 V=800.0 PL=0
MOVL C00795 V=800.0 PL=0
MOVL C00796 V=800.0 PL=0
MOVL C00797 V=800.0 PL=0
MOVL C00798 V=800.0 PL=0
MOVL C00799 V=800.0 PL=0
MOVL C00800 V=800.0 PL=0
MOVL C00801 V=800.0 PL=0
MOVL C00802 V=800.0 PL=0
MOVL C00803 V=800.0 PL=0
MOVL C00804 V=800.0 PL=0
MOVL C00805 V=800.0 PL=0
MOVL C00806 V=800.0 PL=0
MOVL C00807 V=800.0 PL=0
MOVL C00808 V=800.0 PL=0
MOVL C00809 V=800.0 PL=0
MOVL C00810 V=800.0 PL=0
MOVL C00811 V=800.0 PL=0
MOVL C00812 V=800.0 PL=0
MOVL C00813 V=800.0 PL=0
MOVL C00814 V=800.0 PL=0
MOVL C00815 V=800.0 PL=0
MOVL C00816 V=800.0 PL=0
MOVL C00817 V=800.0 PL=0
MOVL C00818 V=800.0 PL=0
MOVL C00819 V=800.0 PL=0
MOVL C00820 V=800.0 PL=0
MOVL C00821 V=800.0 PL=0
MOVL C00822 V=800.0 PL=0
MOVL C00823 V=800.0 PL=0
MOVL C00824 V=800.0 PL=0
MOVL C00825 V=800.0 PL=0
MOVL C00826 V=800.0 PL=0
MOVL C00827 V=800.0 PL=0
MOVL C00828 V=800.0 PL=0
MOVL C00829 V=800.0 PL=0
MOVL C00830 V=800.0 PL=0
MOVL C00831 V=800.0 PL=0
MOVL C00832 V=800.0 PL=0
MOVL C00833 V=800.0 PL=0
MOVL C00834 V=800.0 PL=0
MOVL C00835 V=800.0 PL=0
MOVL C00836 V=800.0 PL=0
MOVL C00837 V=800.0 PL=0
MOVL C00838 V=800.0 PL=0
MOVL C00839 V=800.0 PL=0
MOVL C00840 V=800.0 PL=0
MOVL C00841 V=800.0 PL=0
MOVL C00842 V=800.0 PL=0
MOVL C00843 V=800.0 PL=0
MOVL C00844 V=800.0 PL=0
MOVL C00845 V=800.0 PL=0
MOVL C00846 V=800.0 PL=0
MOVL C00847 V=800.0 PL=0
MOVL C00848 V=800.0 PL=0
MOVL C00849 V=800.0 PL=0
MOVL C00850 V=800.0 PL=0
MOVL C00851 V=800.0 PL=0
MOVL C00852 V=800.0 PL=0
MOVL C00853 V=800.0 PL=0
MOVL C00854 V=800.0 PL=0
MOVL C00855 V=800.0 PL=0
MOVL C00856 V=800.0 PL=0
MOVL C00857 V=800.0 PL=0
MOVL C00858 V=800.0 PL=0
MOVL C00859 V=800.0 PL=0
MOVL C00860 V=800.0 PL=0
MOVL C00861 V=800.0 PL=0
MOVL C00862 V=800.0 PL=0
MOVL C00863 V=800.0 PL=0
MOVL C00864 V=800.0 PL=0
MOVL C00865 V=800.0 PL=0
MOVL C00866 V=800.0 PL=0
MOVL C00867 V=800.0 PL=0
MOVL C00868 V=800.0 PL=0
MOVL C00869 V=800.0 PL=0
MOVL C00870 V=800.0 PL=0
MOVL C00871 V=800.0 PL=0
MOVL C00872 V=800.0 PL=0
MOVL C00873 V=800.0 PL=0
MOVL C00874 V=800.0 PL=0
MOVL C00875 V=800.0 PL=0
MOVL C00876 V=800.0 PL=0
MOVL C00877 V=800.0 PL=0
MOVL C00878 V=800.0 PL=0
MOVL C00879 V=800.0 PL=0
MOVL C00880 V=800.0 PL=0
MOVL C00881 V=800.0 PL=0
MOVL C00882 V=800.0 PL=0
MOVL C00883 V=800.0 PL=0
MOVL C00884 V=800.0 PL=0
MOVL C00885 V=800.0 PL=0
MOVL C00886 V=800.0 PL=0
MOVL C00887 V=800.0 PL=0
MOVL C00888 V=800.0 PL=0
MOVL C00889 V=800.0 PL=0
MOVL C00890 V=800.0 PL=0
MOVL C00891 V=800.0 PL=0
MOVL C00892 V=800.0 PL=0
MOVL C00893 V=800.0 PL=0
MOVL C00894 V=800.0 PL=0
MOVL C00895 V=800.0 PL=0
MOVL C00896 V=800.0 PL=0
MOVL C00897 V=800.0 PL=0
MOVL C00898 V=800.0 PL=0
MOVL C00899 V=800.0 PL=0
MOVL C00900 V=800.0 PL=0
MOVL C00901 V=800.0 PL=0
MOVL C00902 V=800.0 PL=0
MOVL C00903 V=800.0 PL=0
MOVL C00904 V=800.0 PL=0
MOVL C00905 V=800.0 PL=0
MOVL C00906 V=800.0 PL=0
MOVL C00907 V=800.0 PL=0
MOVL C00908 V=800.0 PL=0
MOVL C00909 V=800.0 PL=0
MOVL C00910 V=800.0 PL=0
MOVL C00911 V=800.0 PL=0
MOVL C00912 V=800.0 PL=0
MOVL C00913 V=800.0 PL=0
MOVL C00914 V=800.0 PL=0
MOVL C00915 V=800.0 PL=0
MOVL C00916 V=800.0 PL=0
MOVL C00917 V=800.0 PL=0
MOVL C00918 V=800.0 PL=0
MOVL C00919 V=800.0 PL=0
MOVL C00920 V=800.0 PL=0
MOVL C00921 V=800.0 PL=0
MOVL C00922 V=800.0 PL=0
MOVL C00923 V=800.0 PL=0
MOVL C00924 V=800.0 PL=0
MOVL C00925 V=800.0 PL=0
MOVL C00926 V=800.0 PL=0
MOVL C00927 V=800.0 PL=0
MOVL C00928 V=800.0 PL=0
MOVL C00929 V=800.0 PL=0
MOVL C00930 V=800.0 PL=0
MOVL C00931 V=800.0 PL=0
MOVL C00932 V=800.0 PL=0
MOVL C00933 V=800.0 PL=0
MOVL C00934 V=800.0 PL=0
MOVL C00935 V=800.0 PL=0
MOVL C00936 V=800.0 PL=0
MOVL C00937 V=800.0 PL=0
MOVL C00938 V=800.0 PL=0
MOVL C00939 V=800.0 PL=0
MOVL C00940 V=800.0 PL=0
MOVL C00941 V=800.0 PL=0
MOVL C00942 V=800.0 PL=0
MOVL C00943 V=800.0 PL=0
MOVL C00944 V=800.0 PL=0
MOVL C00945 V=800.0 PL=0
MOVL C00946 V=800.0 PL=0
MOVL C00947 V=800.0 PL=0
MOVL C00948 V=800.0 PL=0
MOVL C00949 V=800.0 PL=0
MOVL C00950 V=800.0 PL=0
MOVL C00951 V=800.0 PL=0
MOVL C00952 V=800.0 PL=0
MOVL C00953 V=800.0 PL=0
MOVL C00954 V=800.0 PL=0
MOVL C00955 V=800.0 PL=0
MOVL C00956 V=800.0 PL=0
MOVL C00957 V=800.0 PL=0
MOVL C00958 V=800.0 PL=0
MOVL C00959 V=800.0 PL=0
MOVL C00960 V=800.0 PL=0
MOVL C00961 V=800.0 PL=0
MOVL C00962 V=800.0 PL=0
MOVL C00963 V=800.0 PL=0
MOVL C00964 V=800.0 PL=0
MOVL C00965 V=800.0 PL=0
MOVL C00966 V=800.0 PL=0
MOVL C00967 V=800.0 PL=0
MOVL C00968 V=800.0 PL=0
MOVL C00969 V=800.0 PL=0
MOVL C00970 V=800.0 PL=0
MOVL C00971 V=800.0 PL=0
MOVL C00972 V=800.0 PL=0
MOVL C00973 V=800.0 PL=0
MOVL C00974 V=800.0 PL=0
MOVL C00975 V=800.0 PL=0
MOVL C00976 V=800.0 PL=0
MOVL C00977 V=800.0 PL=0
MOVL C00978 V=800.0 PL=0
MOVL C00979 V=800.0 PL=0
MOVL C00980 V=800.0 PL=0
MOVL C00981 V=800.0 PL=0
MOVL C00982 V=800.0 PL=0
MOVL C00983 V=800.0 PL=0
MOVL C00984 V=800.0 PL=0
MOVL C00985 V=800.0 PL=0
MOVL C00986 V=800.0 PL=0
MOVL C00987 V=800.0 PL=0
MOVL C00988 V=800.0 PL=0
MOVL C00989 V=800.0 PL=0
MOVL C00990 V=800.0 PL=0
MOVL C00991 V=800.0 PL=0
MOVL C00992 V=800.0 PL=0
MOVL C00993 V=800.0 PL=0
MOVL C00994 V=800.0 PL=0
MOVL C00995 V=800.0 PL=0
MOVL C00996 V=800.0 PL=0
MOVL C00997 V=800.0 PL=0
MOVL C00998 V=800.0 PL=0
MOVL C00999 V=800.0 PL=0
MOVL C01000 V=800.0 PL=0
MOVL C01001 V=800.0 PL=0
MOVL C01002 V=800.0 PL=0
MOVL C01003 V=800.0 PL=0
MOVL C01004 V=800.0 PL=0
MOVL C01005 V=800.0 PL=0
MOVL C01006 V=800.0 PL=0
MOVL C01007 V=800.0 PL=0
MOVL C01008 V=800.0 PL=0
MOVL C01009 V=800.0 PL=0
MOVL C01010 V=800.0 PL=0
MOVL C01011 V=800.0 PL=0
MOVL C01012 V=800.0 PL=0
MOVL C01013 V=800.0 PL=0
MOVL C01014 V=800.0 PL=0
MOVL C01015 V=800.0 PL=0
MOVL C01016 V=800.0 PL=0
MOVL C01017 V=800.0 PL=0
MOVL C01018 V=800.0 PL=0
MOVL C01019 V=800.0 PL=0
MOVL C01020 V=800.0 PL=0
MOVL C01021 V=800.0 PL=0
MOVL C01022 V=800.0 PL=0
MOVL C01023 V=800.0 PL=0
MOVL C01024 V=800.0 PL=0
MOVL C01025 V=800.0 PL=0
MOVL C01026 V=800.0 PL=0
MOVL C01027 V=800.0 PL=0
MOVL C01028 V=800.0 PL=0
MOVL C01029 V=800.0 PL=0
MOVL C01030 V=800.0 PL=0
MOVL C01031 V=800.0 PL=0
MOVL C01032 V=800.0 PL=0
MOVL C01033 V=800.0 PL=0
MOVL C01034 V=800.0 PL=0
MOVL C01035 V=800.0 PL=0
MOVL C01036 V=800.0 PL=0
MOVL C01037 V=800.0 PL=0
MOVL C01038 V=800.0 PL=0
MOVL C01039 V=800.0 PL=0
MOVL C01040 V=800.0 PL=0
MOVL C01041 V=800.0 PL=0
MOVL C01042 V=800.0 PL=0
MOVL C01043 V=800.0 PL=0
MOVL C01044 V=800.0 PL=0
MOVL C01045 V=800.0 PL=0
MOVL C01046 V=800.0 PL=0
MOVL C01047 V=800.0 PL=0
MOVL C01048 V=800.0 PL=0
MOVL C01049 V=800.0 PL=0
MOVL C01050 V=800.0 PL=0
MOVL C01051 V=800.0 PL=0
MOVL C01052 V=800.0 PL=0
MOVL C01053 V=800.0 PL=0
MOVL C01054 V=800.0 PL=0
MOVL C01055 V=800.0 PL=0
MOVL C01056 V=800.0 PL=0
MOVL C01057 V=800.0 PL=0
MOVL C01058 V=800.0 PL=0
MOVL C01059 V=800.0 PL=0
MOVL C01060 V=800.0 PL=0
MOVL C01061 V=800.0 PL=0
MOVL C01062 V=800.0 PL=0
MOVL C01063 V=800.0 PL=0
MOVL C01064 V=800.0 PL=0
MOVL C01065 V=800.0 PL=0
MOVL C01066 V=800.0 PL=0
MOVL C01067 V=800.0 PL=0
MOVL C01068 V=800.0 PL=0
MOVL C01069 V=800.0 PL=0
MOVL C01070 V=800.0 PL=0
MOVL C01071 V=800.0 PL=0
MOVL C01072 V=800.0 PL=0
MOVL C01073 V=800.0 PL=0
MOVL C01074 V=800.0 PL=0
MOVL C01075 V=800.0 PL=0
MOVL C01076 V=800.0 PL=0
MOVL C01077 V=800.0 PL=0
MOVL C01078 V=800.0 PL=0
MOVL C01079 V=800.0 PL=0
MOVL C01080 V=800.0 PL=0
MOVL C01081 V=800.0 PL=0
MOVL C01082 V=800.0 PL=0
MOVL C01083 V=800.0 PL=0
MOVL C01084 V=800.0 PL=0
MOVL C01085 V=800.0 PL=0
MOVL C01086 V=800.0 PL=0
MOVL C01087 V=800.0 PL=0
MOVL C01088 V=800.0 PL=0
MOVL C01089 V=800.0 PL=0
MOVL C01090 V=800.0 PL=0
MOVL C01091 V=800.0 PL=0
MOVL C01092 V=800.0 PL=0
MOVL C01093 V=800.0 PL=0
MOVL C01094 V=800.0 PL=0
MOVL C01095 V=800.0 PL=0
MOVL C01096 V=800.0 PL=0
MOVL C01097 V=800.0 PL=0
MOVL C01098 V=800.0 PL=0
MOVL C01099 V=800.0 PL=0
MOVL C01100 V=800.0 PL=0
MOVL C01101 V=800.0 PL=0
MOVL C01102 V=800.0 PL=0
MOVL C01103 V=800.0 PL=0
MOVL C01104 V=800.0 PL=0
MOVL C01105 V=800.0 PL=0
MOVL C01106 V=800.0 PL=0
MOVL C01107 V=800.0 PL=0
MOVL C01108 V=800.0 PL=0
MOVL C01109 V=800.0 PL=0
MOVL C01110 V=800.0 PL=0
MOVL C01111 V=800.0 PL=0
MOVL C01112 V=800.0 PL=0
MOVL C01113 V=800.0 PL=0
MOVL C01114 V=800.0 PL=0
MOVL C01115 V=800.0 PL=0
MOVL C01116 V=800.0 PL=0
MOVL C01117 V=800.0 PL=0
MOVL C01118 V=800.0 PL=0
MOVL C01119 V=800.0 PL=0
MOVL C01120 V=800.0 PL=0
MOVL C01121 V=800.0 PL=0
MOVL C01122 V=800.0 PL=0
MOVL C01123 V=800.0 PL=0
MOVL C01124 V=800.0 PL=0
MOVL C01125 V=800.0 PL=0
MOVL C01126 V=800.0 PL=0
MOVL C01127 V=800.0 PL=0
MOVL C01128 V=800.0 PL=0
MOVL C01129 V=800.0 PL=0
MOVL C01130 V=800.0 PL=0
MOVL C01131 V=800.0 PL=0
MOVL C01132 V=800.0 PL=0
MOVL C01133 V=800.0 PL=0
MOVL C01134 V=800.0 PL=0
MOVL C01135 V=800.0 PL=0
MOVL C01136 V=800.0 PL=0
MOVL C01137 V=800.0 PL=0
MOVL C01138 V=800.0 PL=0
MOVL C01139 V=800.0 PL=0
MOVL C01140 V=800.0 PL=0
MOVL C01141 V=800.0 PL=0
MOVL C01142 V=800.0 PL=0
MOVL C01143 V=800.0 PL=0
MOVL C01144 V=800.0 PL=0
MOVL C01145 V=800.0 PL=0
MOVL C01146 V=800.0 PL=0
MOVL C01147 V=800.0 PL=0
MOVL C01148 V=800.0 PL=0
MOVL C01149 V=800.0 PL=0
MOVL C01150 V=800.0 PL=0
MOVL C01151 V=800.0 PL=0
MOVL C01152 V=800.0 PL=0
MOVL C01153 V=800.0 PL=0
MOVL C01154 V=800.0 PL=0
MOVL C01155 V=800.0 PL=0
MOVL C01156 V=800.0 PL=0
MOVL C01157 V=800.0 PL=0
MOVL C01158 V=800.0 PL=0
MOVL C01159 V=800.0 PL=0
MOVL C01160 V=800.0 PL=0
MOVL C01161 V=800.0 PL=0
MOVL C01162 V=800.0 PL=0
MOVL C01163 V=800.0 PL=0
MOVL C01164 V=800.0 PL=0
MOVL C01165 V=800.0 PL=0
MOVL C01166 V=800.0 PL=0
MOVL C01167 V=800.0 PL=0
MOVL C01168 V=800.0 PL=0
MOVL C01169 V=800.0 PL=0
MOVL C01170 V=800.0 PL=0
MOVL C01171 V=800.0 PL=0
MOVL C01172 V=800.0 PL=0
MOVL C01173 V=800.0 PL=0
MOVL C01174 V=800.0 PL=0
MOVL C01175 V=800.0 PL=0
MOVL C01176 V=800.0 PL=0
MOVL C01177 V=800.0 PL=0
MOVL C01178 V=800.0 PL=0
MOVL C01179 V=800.0 PL=0
MOVL C01180 V=800.0 PL=0
MOVL C01181 V=800.0 PL=0
MOVL C01182 V=800.0 PL=0
MOVL C01183 V=800.0 PL=0
MOVL C01184 V=800.0 PL=0
MOVL C01185 V=800.0 PL=0
MOVL C01186 V=800.0 PL=0
MOVL C01187 V=800.0 PL=0
MOVL C01188 V=800.0 PL=0
MOVL C01189 V=800.0 PL=0
MOVL C01190 V=800.0 PL=0
MOVL C01191 V=800.0 PL=0
MOVL C01192 V=800.0 PL=0
MOVL C01193 V=800.0 PL=0
MOVL C01194 V=800.0 PL=0
MOVL C01195 V=800.0 PL=0
MOVL C01196 V=800.0 PL=0
MOVL C01197 V=800.0 PL=0
MOVL C01198 V=800.0 PL=0
MOVL C01199 V=800.0 PL=0
MOVL C01200 V=800.0 PL=0
MOVL C01201 V=800.0 PL=0
MOVL C01202 V=800.0 PL=0
MOVL C01203 V=800.0 PL=0
MOVL C01204 V=800.0 PL=0
MOVL C01205 V=800.0 PL=0
MOVL C01206 V=800.0 PL=0
MOVL C01207 V=800.0 PL=0
MOVL C01208 V=800.0 PL=0
MOVL C01209 V=800.0 PL=0
MOVL C01210 V=800.0 PL=0
MOVL C01211 V=800.0 PL=0
MOVL C01212 V=800.0 PL=0
MOVL C01213 V=800.0 PL=0
MOVL C01214 V=800.0 PL=0
MOVL C01215 V=800.0 PL=0
MOVL C01216 V=800.0 PL=0
MOVL C01217 V=800.0 PL=0
MOVL C01218 V=800.0 PL=0
MOVL C01219 V=800.0 PL=0
MOVL C01220 V=800.0 PL=0
MOVL C01221 V=800.0 PL=0
MOVL C01222 V=800.0 PL=0
MOVL C01223 V=800.0 PL=0
MOVL C01224 V=800.0 PL=0
MOVL C01225 V=800.0 PL=0
MOVL C01226 V=800.0 PL=0
MOVL C01227 V=800.0 PL=0
MOVL C01228 V=800.0 PL=0
MOVL C01229 V=800.0 PL=0
MOVL C01230 V=800.0 PL=0
MOVL C01231 V=800.0 PL=0
MOVL C01232 V=800.0 PL=0
MOVL C01233 V=800.0 PL=0
MOVL C01234 V=800.0 PL=0
MOVL C01235 V=800.0 PL=0
MOVL C01236 V=800.0 PL=0
MOVL C01237 V=800.0 PL=0
MOVL C01238 V=800.0 PL=0
MOVL C01239 V=800.0 PL=0
MOVL C01240 V=800.0 PL=0
MOVL C01241 V=800.0 PL=0
MOVL C01242 V=800.0 PL=0
MOVL C01243 V=800.0 PL=0
MOVL C01244 V=800.0 PL=0
MOVL C01245 V=800.0 PL=0
MOVL C01246 V=800.0 PL=0
MOVL C01247 V=800.0 PL=0
MOVL C01248 V=800.0 PL=0
MOVL C01249 V=800.0 PL=0
MOVL C01250 V=800.0 PL=0
MOVL C01251 V=800.0 PL=0
MOVL C01252 V=800.0 PL=0
MOVL C01253 V=800.0 PL=0
MOVL C01254 V=800.0 PL=0
MOVL C01255 V=800.0 PL=0
MOVL C01256 V=800.0 PL=0
MOVL C01257 V=800.0 PL=0
MOVL C01258 V=800.0 PL=0
MOVL C01259 V=800.0 PL=0
MOVL C01260 V=800.0 PL=0
MOVL C01261 V=800.0 PL=0
MOVL C01262 V=800.0 PL=0
MOVL C01263 V=800.0 PL=0
MOVL C01264 V=800.0 PL=0
MOVL C01265 V=800.0 PL=0
MOVL C01266 V=800.0 PL=0
MOVL C01267 V=800.0 PL=0
MOVL C01268 V=800.0 PL=0
MOVL C01269 V=800.0 PL=0
MOVL C01270 V=800.0 PL=0
MOVL C01271 V=800.0 PL=0
MOVL C01272 V=800.0 PL=0
MOVL C01273 V=800.0 PL=0
MOVL C01274 V=800.0 PL=0
MOVL C01275 V=800.0 PL=0
MOVL C01276 V=800.0 PL=0
MOVL C01277 V=800.0 PL=0
MOVL C01278 V=800.0 PL=0
MOVL C01279 V=800.0 PL=0
MOVL C01280 V=800.0 PL=0
MOVL C01281 V=800.0 PL=0
MOVL C01282 V=800.0 PL=0
MOVL C01283 V=800.0 PL=0
MOVL C01284 V=800.0 PL=0
MOVL C01285 V=800.0 PL=0
MOVL C01286 V=800.0 PL=0
MOVL C01287 V=800.0 PL=0
MOVL C01288 V=800.0 PL=0
MOVL C01289 V=800.0 PL=0
MOVL C01290 V=800.0 PL=0
MOVL C01291 V=800.0 PL=0
MOVL C01292 V=800.0 PL=0
MOVL C01293 V=800.0 PL=0
MOVL C01294 V=800.0 PL=0
MOVL C01295 V=800.0 PL=0
MOVL C01296 V=800.0 PL=0
MOVL C01297 V=800.0 PL=0
MOVL C01298 V=800.0 PL=0
MOVL C01299 V=800.0 PL=0
MOVL C01300 V=800.0 PL=0
MOVL C01301 V=800.0 PL=0
MOVL C01302 V=800.0 PL=0
MOVL C01303 V=800.0 PL=0
MOVL C01304 V=800.0 PL=0
MOVL C01305 V=800.0 PL=0
MOVL C01306 V=800.0 PL=0
MOVL C01307 V=800.0 PL=0
MOVL C01308 V=800.0 PL=0
MOVL C01309 V=800.0 PL=0
MOVL C01310 V=800.0 PL=0
MOVL C01311 V=800.0 PL=0
MOVL C01312 V=800.0 PL=0
MOVL C01313 V=800.0 PL=0
MOVL C01314 V=800.0 PL=0
MOVL C01315 V=800.0 PL=0
MOVL C01316 V=800.0 PL=0
MOVL C01317 V=800.0 PL=0
MOVL C01318 V=800.0 PL=0
MOVL C01319 V=800.0 PL=0
MOVL C01320 V=800.0 PL=0
MOVL C01321 V=800.0 PL=0
MOVL C01322 V=800.0 PL=0
MOVL C01323 V=800.0 PL=0
MOVL C01324 V=800.0 PL=0
MOVL C01325 V=800.0 PL=0
MOVL C01326 V=800.0 PL=0
MOVL C01327 V=800.0 PL=0
MOVL C01328 V=800.0 PL=0
MOVL C01329 V=800.0 PL=0
MOVL C01330 V=800.0 PL=0
MOVL C01331 V=800.0 PL=0
MOVL C01332 V=800.0 PL=0
MOVL C01333 V=800.0 PL=0
MOVL C01334 V=800.0 PL=0
MOVL C01335 V=800.0 PL=0
MOVL C01336 V=800.0 PL=0
MOVL C01337 V=800.0 PL=0
MOVL C01338 V=800.0 PL=0
MOVL C01339 V=800.0 PL=0
MOVL C01340 V=800.0 PL=0
MOVL C01341 V=800.0 PL=0
MOVL C01342 V=800.0 PL=0
MOVL C01343 V=800.0 PL=0
MOVL C01344 V=800.0 PL=0
MOVL C01345 V=800.0 PL=0
MOVL C01346 V=800.0 PL=0
MOVL C01347 V=800.0 PL=0
MOVL C01348 V=800.0 PL=0
MOVL C01349 V=800.0 PL=0
MOVL C01350 V=800.0 PL=0
MOVL C01351 V=800.0 PL=0
MOVL C01352 V=800.0 PL=0
MOVL C01353 V=800.0 PL=0
MOVL C01354 V=800.0 PL=0
MOVL C01355 V=800.0 PL=0
MOVL C01356 V=800.0 PL=0
MOVL C01357 V=800.0 PL=0
MOVL C01358 V=800.0 PL=0
MOVL C01359 V=800.0 PL=0
MOVL C01360 V=800.0 PL=0
MOVL C01361 V=800.0 PL=0
MOVL C01362 V=800.0 PL=0
MOVL C01363 V=800.0 PL=0
MOVL C01364 V=800.0 PL=0
MOVL C01365 V=800.0 PL=0
MOVL C01366 V=800.0 PL=0
MOVL C01367 V=800.0 PL=0
MOVL C01368 V=800.0 PL=0
MOVL C01369 V=800.0 PL=0
MOVL C01370 V=800.0 PL=0
MOVL C01371 V=800.0 PL=0
MOVL C01372 V=800.0 PL=0
MOVL C01373 V=800.0 PL=0
MOVL C01374 V=800.0 PL=0
MOVL C01375 V=800.0 PL=0
MOVL C01376 V=800.0 PL=0
MOVL C01377 V=800.0 PL=0
MOVL C01378 V=800.0 PL=0
MOVL C01379 V=800.0 PL=0
MOVL C01380 V=800.0 PL=0
MOVL C01381 V=800.0 PL=0
MOVL C01382 V=800.0 PL=0
MOVL C01383 V=800.0 PL=0
MOVL C01384 V=800.0 PL=0
MOVL C01385 V=800.0 PL=0
MOVL C01386 V=800.0 PL=0
MOVL C01387 V=800.0 PL=0
MOVL C01388 V=800.0 PL=0
MOVL C01389 V=800.0 PL=0
MOVL C01390 V=800.0 PL=0
MOVL C01391 V=800.0 PL=0
MOVL C01392 V=800.0 PL=0
MOVL C01393 V=800.0 PL=0
MOVL C01394 V=800.0 PL=0
MOVL C01395 V=800.0 PL=0
MOVL C01396 V=800.0 PL=0
MOVL C01397 V=800.0 PL=0
MOVL C01398 V=800.0 PL=0
MOVL C01399 V=800.0 PL=0
MOVL C01400 V=800.0 PL=0
MOVL C01401 V=800.0 PL=0
MOVL C01402 V=800.0 PL=0
MOVL C01403 V=800.0 PL=0
MOVL C01404 V=800.0 PL=0
MOVL C01405 V=800.0 PL=0
MOVL C01406 V=800.0 PL=0
MOVL C01407 V=800.0 PL=0
MOVL C01408 V=800.0 PL=0
MOVL C01409 V=800.0 PL=0
MOVL C01410 V=800.0 PL=0
MOVL C01411 V=800.0 PL=0
MOVL C01412 V=800.0 PL=0
MOVL C01413 V=800.0 PL=0
MOVL C01414 V=800.0 PL=0
MOVL C01415 V=800.0 PL=0
MOVL C01416 V=800.0 PL=0
MOVL C01417 V=800.0 PL=0
MOVL C01418 V=800.0 PL=0
MOVL C01419 V=800.0 PL=0
MOVL C01420 V=800.0 PL=0
MOVL C01421 V=800.0 PL=0
MOVL C01422 V=800.0 PL=0
MOVL C01423 V=800.0 PL=0
MOVL C01424 V=800.0 PL=0
MOVL C01425 V=800.0 PL=0
MOVL C01426 V=800.0 PL=0
MOVL C01427 V=800.0 PL=0
MOVL C01428 V=800.0 PL=0
MOVL C01429 V=800.0 PL=0
MOVL C01430 V=800.0 PL=0
MOVL C01431 V=800.0 PL=0
MOVL C01432 V=800.0 PL=0
MOVL C01433 V=800.0 PL=0
MOVL C01434 V=800.0 PL=0
MOVL C01435 V=800.0 PL=0
MOVL C01436 V=800.0 PL=0
MOVL C01437 V=800.0 PL=0
MOVL C01438 V=800.0 PL=0
MOVL C01439 V=800.0 PL=0
MOVL C01440 V=800.0 PL=0
MOVL C01441 V=800.0 PL=0
MOVL C01442 V=800.0 PL=0
MOVL C01443 V=800.0 PL=0
MOVL C01444 V=800.0 PL=0
MOVL C01445 V=800.0 PL=0
MOVL C01446 V=800.0 PL=0
MOVL C01447 V=800.0 PL=0
MOVL C01448 V=800.0 PL=0
MOVL C01449 V=800.0 PL=0
MOVL C01450 V=800.0 PL=0
MOVL C01451 V=800.0 PL=0
MOVL C01452 V=800.0 PL=0
MOVL C01453 V=800.0 PL=0
MOVL C01454 V=800.0 PL=0
MOVL C01455 V=800.0 PL=0
MOVL C01456 V=800.0 PL=0
MOVL C01457 V=800.0 PL=0
MOVL C01458 V=800.0 PL=0
MOVL C01459 V=800.0 PL=0
MOVL C01460 V=800.0 PL=0
MOVL C01461 V=800.0 PL=0
MOVL C01462 V=800.0 PL=0
MOVL C01463 V=800.0 PL=0
MOVL C01464 V=800.0 PL=0
MOVL C01465 V=800.0 PL=0
MOVL C01466 V=800.0 PL=0
MOVL C01467 V=800.0 PL=0
MOVL C01468 V=800.0 PL=0
MOVL C01469 V=800.0 PL=0
MOVL C01470 V=800.0 PL=0
MOVL C01471 V=800.0 PL=0
MOVL C01472 V=800.0 PL=0
MOVL C01473 V=800.0 PL=0
MOVL C01474 V=800.0 PL=0
MOVL C01475 V=800.0 PL=0
MOVL C01476 V=800.0 PL=0
MOVL C01477 V=800.0 PL=0
MOVL C01478 V=800.0 PL=0
MOVL C01479 V=800.0 PL=0
MOVL C01480 V=800.0 PL=0
MOVL C01481 V=800.0 PL=0
MOVL C01482 V=800.0 PL=0
MOVL C01483 V=800.0 PL=0
MOVL C01484 V=800.0 PL=0
MOVL C01485 V=800.0 PL=0
MOVL C01486 V=800.0 PL=0
MOVL C01487 V=800.0 PL=0
MOVL C01488 V=800.0 PL=0
MOVL C01489 V=800.0 PL=0
MOVL C01490 V=800.0 PL=0
MOVL C01491 V=800.0 PL=0
MOVL C01492 V=800.0 PL=0
MOVL C01493 V=800.0 PL=0
MOVL C01494 V=800.0 PL=0
MOVL C01495 V=800.0 PL=0
MOVL C01496 V=800.0 PL=0
MOVL C01497 V=800.0 PL=0
MOVL C01498 V=800.0 PL=0
MOVL C01499 V=800.0 PL=0
MOVL C01500 V=800.0 PL=0
MOVL C01501 V=800.0 PL=0
MOVL C01502 V=800.0 PL=0
MOVL C01503 V=800.0 PL=0
MOVL C01504 V=800.0 PL=0
MOVL C01505 V=800.0 PL=0
MOVL C01506 V=800.0 PL=0
MOVL C01507 V=800.0 PL=0
MOVL C01508 V=800.0 PL=0
MOVL C01509 V=800.0 PL=0
MOVL C01510 V=800.0 PL=0
MOVL C01511 V=800.0 PL=0
MOVL C01512 V=800.0 PL=0
MOVL C01513 V=800.0 PL=0
MOVL C01514 V=800.0 PL=0
MOVL C01515 V=800.0 PL=0
MOVL C01516 V=800.0 PL=0
MOVL C01517 V=800.0 PL=0
MOVL C01518 V=800.0 PL=0
MOVL C01519 V=800.0 PL=0
MOVL C01520 V=800.0 PL=0
MOVL C01521 V=800.0 PL=0
MOVL C01522 V=800.0 PL=0
MOVL C01523 V=800.0 PL=0
MOVL C01524 V=800.0 PL=0
MOVL C01525 V=800.0 PL=0
MOVL C01526 V=800.0 PL=0
MOVL C01527 V=800.0 PL=0
MOVL C01528 V=800.0 PL=0
MOVL C01529 V=800.0 PL=0
MOVL C01530 V=800.0 PL=0
MOVL C01531 V=800.0 PL=0
MOVL C01532 V=800.0 PL=0
MOVL C01533 V=800.0 PL=0
MOVL C01534 V=800.0 PL=0
MOVL C01535 V=800.0 PL=0
MOVL C01536 V=800.0 PL=0
MOVL C01537 V=800.0 PL=0
MOVL C01538 V=800.0 PL=0
MOVL C01539 V=800.0 PL=0
MOVL C01540 V=800.0 PL=0
MOVL C01541 V=800.0 PL=0
MOVL C01542 V=800.0 PL=0
MOVL C01543 V=800.0 PL=0
MOVL C01544 V=800.0 PL=0
MOVL C01545 V=800.0 PL=0
MOVL C01546 V=800.0 PL=0
MOVL C01547 V=800.0 PL=0
MOVL C01548 V=800.0 PL=0
MOVL C01549 V=800.0 PL=0
MOVL C01550 V=800.0 PL=0
MOVL C01551 V=800.0 PL=0
MOVL C01552 V=800.0 PL=0
MOVL C01553 V=800.0 PL=0
MOVL C01554 V=800.0 PL=0
MOVL C01555 V=800.0 PL=0
MOVL C01556 V=800.0 PL=0
MOVL C01557 V=800.0 PL=0
MOVL C01558 V=800.0 PL=0
MOVL C01559 V=800.0 PL=0
MOVL C01560 V=800.0 PL=0
MOVL C01561 V=800.0 PL=0
MOVL C01562 V=800.0 PL=0
MOVL C01563 V=800.0 PL=0
MOVL C01564 V=800.0 PL=0
MOVL C01565 V=800.0 PL=0
MOVL C01566 V=800.0 PL=0
MOVL C01567 V=800.0 PL=0
MOVL C01568 V=800.0 PL=0
MOVL C01569 V=800.0 PL=0
MOVL C01570 V=800.0 PL=0
MOVL C01571 V=800.0 PL=0
MOVL C01572 V=800.0 PL=0
MOVL C01573 V=800.0 PL=0
MOVL C01574 V=800.0 PL=0
MOVL C01575 V=800.0 PL=0
MOVL C01576 V=800.0 PL=0
MOVL C01577 V=800.0 PL=0
MOVL C01578 V=800.0 PL=0
MOVL C01579 V=800.0 PL=0
MOVL C01580 V=800.0 PL=0
MOVL C01581 V=800.0 PL=0
MOVL C01582 V=800.0 PL=0
MOVL C01583 V=800.0 PL=0
MOVL C01584 V=800.0 PL=0
MOVL C01585 V=800.0 PL=0
MOVL C01586 V=800.0 PL=0
MOVL C01587 V=800.0 PL=0
MOVL C01588 V=800.0 PL=0
MOVL C01589 V=800.0 PL=0
MOVL C01590 V=800.0 PL=0
MOVL C01591 V=800.0 PL=0
MOVL C01592 V=800.0 PL=0
MOVL C01593 V=800.0 PL=0
MOVL C01594 V=800.0 PL=0
MOVL C01595 V=800.0 PL=0
MOVL C01596 V=800.0 PL=0
MOVL C01597 V=800.0 PL=0
MOVL C01598 V=800.0 PL=0
MOVL C01599 V=800.0 PL=0
MOVL C01600 V=800.0 PL=0
MOVL C01601 V=800.0 PL=0
MOVL C01602 V=800.0 PL=0
MOVL C01603 V=800.0 PL=0
MOVL C01604 V=800.0 PL=0
MOVL C01605 V=800.0 PL=0
MOVL C01606 V=800.0 PL=0
MOVL C01607 V=800.0 PL=0
MOVL C01608 V=800.0 PL=0
MOVL C01609 V=800.0 PL=0
MOVL C01610 V=800.0 PL=0
MOVL C01611 V=800.0 PL=0
MOVL C01612 V=800.0 PL=0
MOVL C01613 V=800.0 PL=0
MOVL C01614 V=800.0 PL=0
MOVL C01615 V=800.0 PL=0
MOVL C01616 V=800.0 PL=0
MOVL C01617 V=800.0 PL=0
MOVL C01618 V=800.0 PL=0
MOVL C01619 V=800.0 PL=0
MOVL C01620 V=800.0 PL=0
MOVL C01621 V=800.0 PL=0
MOVL C01622 V=800.0 PL=0
MOVL C01623 V=800.0 PL=0
MOVL C01624 V=800.0 PL=0
MOVL C01625 V=800.0 PL=0
MOVL C01626 V=800.0 PL=0
MOVL C01627 V=800.0 PL=0
MOVL C01628 V=800.0 PL=0
MOVL C01629 V=800.0 PL=0
MOVL C01630 V=800.0 PL=0
MOVL C01631 V=800.0 PL=0
MOVL C01632 V=800.0 PL=0
MOVL C01633 V=800.0 PL=0
MOVL C01634 V=800.0 PL=0
MOVL C01635 V=800.0 PL=0
MOVL C01636 V=800.0 PL=0
MOVL C01637 V=800.0 PL=0
MOVL C01638 V=800.0 PL=0
MOVL C01639 V=800.0 PL=0
MOVL C01640 V=800.0 PL=0
MOVL C01641 V=800.0 PL=0
MOVL C01642 V=800.0 PL=0
MOVL C01643 V=800.0 PL=0
MOVL C01644 V=800.0 PL=0
MOVL C01645 V=800.0 PL=0
MOVL C01646 V=800.0 PL=0
MOVL C01647 V=800.0 PL=0
MOVL C01648 V=800.0 PL=0
MOVL C01649 V=800.0 PL=0
MOVL C01650 V=800.0 PL=0
MOVL C01651 V=800.0 PL=0
MOVL C01652 V=800.0 PL=0
MOVL C01653 V=800.0 PL=0
MOVL C01654 V=800.0 PL=0
MOVL C01655 V=800.0 PL=0
MOVL C01656 V=800.0 PL=0
MOVL C01657 V=800.0 PL=0
MOVL C01658 V=800.0 PL=0
MOVL C01659 V=800.0 PL=0
MOVL C01660 V=800.0 PL=0
MOVL C01661 V=800.0 PL=0
MOVL C01662 V=800.0 PL=0
MOVL C01663 V=800.0 PL=0
MOVL C01664 V=800.0 PL=0
MOVL C01665 V=800.0 PL=0
MOVL C01666 V=800.0 PL=0
MOVL C01667 V=800.0 PL=0
MOVL C01668 V=800.0 PL=0
MOVL C01669 V=800.0 PL=0
MOVL C01670 V=800.0 PL=0
MOVL C01671 V=800.0 PL=0
MOVL C01672 V=800.0 PL=0
MOVL C01673 V=800.0 PL=0
MOVL C01674 V=800.0 PL=0
MOVL C01675 V=800.0 PL=0
MOVL C01676 V=800.0 PL=0
MOVL C01677 V=800.0 PL=0
MOVL C01678 V=800.0 PL=0
MOVL C01679 V=800.0 PL=0
MOVL C01680 V=800.0 PL=0
MOVL C01681 V=800.0 PL=0
MOVL C01682 V=800.0 PL=0
MOVL C01683 V=800.0 PL=0
MOVL C01684 V=800.0 PL=0
MOVL C01685 V=800.0 PL=0
MOVL C01686 V=800.0 PL=0
MOVL C01687 V=800.0 PL=0
MOVL C01688 V=800.0 PL=0
MOVL C01689 V=800.0 PL=0
MOVL C01690 V=800.0 PL=0
MOVL C01691 V=800.0 PL=0
MOVL C01692 V=800.0 PL=0
MOVL C01693 V=800.0 PL=0
MOVL C01694 V=800.0 PL=0
MOVL C01695 V=800.0 PL=0
MOVL C01696 V=800.0 PL=0
MOVL C01697 V=800.0 PL=0
MOVL C01698 V=800.0 PL=0
MOVL C01699 V=800.0 PL=0
MOVL C01700 V=800.0 PL=0
MOVL C01701 V=800.0 PL=0
MOVL C01702 V=800.0 PL=0
MOVL C01703 V=800.0 PL=0
MOVL C01704 V=800.0 PL=0
MOVL C01705 V=800.0 PL=0
MOVL C01706 V=800.0 PL=0
MOVL C01707 V=800.0 PL=0
MOVL C01708 V=800.0 PL=0
MOVL C01709 V=800.0 PL=0
MOVL C01710 V=800.0 PL=0
MOVL C01711 V=800.0 PL=0
MOVL C01712 V=800.0 PL=0
MOVL C01713 V=800.0 PL=0
MOVL C01714 V=800.0 PL=0
MOVL C01715 V=800.0 PL=0
MOVL C01716 V=800.0 PL=0
MOVL C01717 V=800.0 PL=0
MOVL C01718 V=800.0 PL=0
MOVL C01719 V=800.0 PL=0
MOVL C01720 V=800.0 PL=0
MOVL C01721 V=800.0 PL=0
MOVL C01722 V=800.0 PL=0
MOVL C01723 V=800.0 PL=0
MOVL C01724 V=800.0 PL=0
MOVL C01725 V=800.0 PL=0
MOVL C01726 V=800.0 PL=0
MOVL C01727 V=800.0 PL=0
MOVL C01728 V=800.0 PL=0
MOVL C01729 V=800.0 PL=0
MOVL C01730 V=800.0 PL=0
MOVL C01731 V=800.0 PL=0
MOVL C01732 V=800.0 PL=0
MOVL C01733 V=800.0 PL=0
MOVL C01734 V=800.0 PL=0
MOVL C01735 V=800.0 PL=0
MOVL C01736 V=800.0 PL=0
MOVL C01737 V=800.0 PL=0
MOVL C01738 V=800.0 PL=0
MOVL C01739 V=800.0 PL=0
MOVL C01740 V=800.0 PL=0
MOVL C01741 V=800.0 PL=0
MOVL C01742 V=800.0 PL=0
MOVL C01743 V=800.0 PL=0
MOVL C01744 V=800.0 PL=0
MOVL C01745 V=800.0 PL=0
MOVL C01746 V=800.0 PL=0
MOVL C01747 V=800.0 PL=0
MOVL C01748 V=800.0 PL=0
MOVL C01749 V=800.0 PL=0
MOVL C01750 V=800.0 PL=0
MOVL C01751 V=800.0 PL=0
MOVL C01752 V=800.0 PL=0
MOVL C01753 V=800.0 PL=0
MOVL C01754 V=800.0 PL=0
MOVL C01755 V=800.0 PL=0
MOVL C01756 V=800.0 PL=0
MOVL C01757 V=800.0 PL=0
MOVL C01758 V=800.0 PL=0
MOVL C01759 V=800.0 PL=0
MOVL C01760 V=800.0 PL=0
MOVL C01761 V=800.0 PL=0
MOVL C01762 V=800.0 PL=0
MOVL C01763 V=800.0 PL=0
MOVL C01764 V=800.0 PL=0
MOVL C01765 V=800.0 PL=0
MOVL C01766 V=800.0 PL=0
MOVL C01767 V=800.0 PL=0
MOVL C01768 V=800.0 PL=0
MOVL C01769 V=800.0 PL=0
MOVL C01770 V=800.0 PL=0
MOVL C01771 V=800.0 PL=0
MOVL C01772 V=800.0 PL=0
MOVL C01773 V=800.0 PL=0
MOVL C01774 V=800.0 PL=0
MOVL C01775 V=800.0 PL=0
MOVL C01776 V=800.0 PL=0
MOVL C01777 V=800.0 PL=0
MOVL C01778 V=800.0 PL=0
MOVL C01779 V=800.0 PL=0
MOVL C01780 V=800.0 PL=0
MOVL C01781 V=800.0 PL=0
MOVL C01782 V=800.0 PL=0
MOVL C01783 V=800.0 PL=0
MOVL C01784 V=800.0 PL=0
MOVL C01785 V=800.0 PL=0
MOVL C01786 V=800.0 PL=0
MOVL C01787 V=800.0 PL=0
MOVL C01788 V=800.0 PL=0
MOVL C01789 V=800.0 PL=0
MOVL C01790 V=800.0 PL=0
MOVL C01791 V=800.0 PL=0
MOVL C01792 V=800.0 PL=0
MOVL C01793 V=800.0 PL=0
MOVL C01794 V=800.0 PL=0
MOVL C01795 V=800.0 PL=0
MOVL C01796 V=800.0 PL=0
MOVL C01797 V=800.0 PL=0
MOVL C01798 V=800.0 PL=0
MOVL C01799 V=800.0 PL=0
MOVL C01800 V=800.0 PL=0
MOVL C01801 V=800.0 PL=0
MOVL C01802 V=800.0 PL=0
MOVL C01803 V=800.0 PL=0
MOVL C01804 V=800.0 PL=0
MOVL C01805 V=800.0 PL=0
MOVL C01806 V=800.0 PL=0
MOVL C01807 V=800.0 PL=0
MOVL C01808 V=800.0 PL=0
MOVL C01809 V=800.0 PL=0
MOVL C01810 V=800.0 PL=0
MOVL C01811 V=800.0 PL=0
MOVL C01812 V=800.0 PL=0
MOVL C01813 V=800.0 PL=0
MOVL C01814 V=800.0 PL=0
MOVL C01815 V=800.0 PL=0
MOVL C01816 V=800.0 PL=0
MOVL C01817 V=800.0 PL=0
MOVL C01818 V=800.0 PL=0
MOVL C01819 V=800.0 PL=0
MOVL C01820 V=800.0 PL=0
MOVL C01821 V=800.0 PL=0
MOVL C01822 V=800.0 PL=0
MOVL C01823 V=800.0 PL=0
MOVL C01824 V=800.0 PL=0
MOVL C01825 V=800.0 PL=0
MOVL C01826 V=800.0 PL=0
MOVL C01827 V=800.0 PL=0
MOVL C01828 V=800.0 PL=0
MOVL C01829 V=800.0 PL=0
MOVL C01830 V=800.0 PL=0
MOVL C01831 V=800.0 PL=0
MOVL C01832 V=800.0 PL=0
MOVL C01833 V=800.0 PL=0
MOVL C01834 V=800.0 PL=0
MOVL C01835 V=800.0 PL=0
MOVL C01836 V=800.0 PL=0
MOVL C01837 V=800.0 PL=0
MOVL C01838 V=800.0 PL=0
MOVL C01839 V=800.0 PL=0
MOVL C01840 V=800.0 PL=0
MOVL C01841 V=800.0 PL=0
MOVL C01842 V=800.0 PL=0
MOVL C01843 V=800.0 PL=0
MOVL C01844 V=800.0 PL=0
MOVL C01845 V=800.0 PL=0
MOVL C01846 V=800.0 PL=0
MOVL C01847 V=800.0 PL=0
MOVL C01848 V=800.0 PL=0
MOVL C01849 V=800.0 PL=0
MOVL C01850 V=800.0 PL=0
MOVL C01851 V=800.0 PL=0
MOVL C01852 V=800.0 PL=0
MOVL C01853 V=800.0 PL=0
MOVL C01854 V=800.0 PL=0
MOVL C01855 V=800.0 PL=0
MOVL C01856 V=800.0 PL=0
MOVL C01857 V=800.0 PL=0
MOVL C01858 V=800.0 PL=0
MOVL C01859 V=800.0 PL=0
MOVL C01860 V=800.0 PL=0
MOVL C01861 V=800.0 PL=0
MOVL C01862 V=800.0 PL=0
MOVL C01863 V=800.0 PL=0
MOVL C01864 V=800.0 PL=0
MOVL C01865 V=800.0 PL=0
MOVL C01866 V=800.0 PL=0
MOVL C01867 V=800.0 PL=0
MOVL C01868 V=800.0 PL=0
MOVL C01869 V=800.0 PL=0
MOVL C01870 V=800.0 PL=0
MOVL C01871 V=800.0 PL=0
MOVL C01872 V=800.0 PL=0
MOVL C01873 V=800.0 PL=0
MOVL C01874 V=800.0 PL=0
MOVL C01875 V=800.0 PL=0
MOVL C01876 V=800.0 PL=0
MOVL C01877 V=800.0 PL=0
MOVL C01878 V=800.0 PL=0
MOVL C01879 V=800.0 PL=0
MOVL C01880 V=800.0 PL=0
MOVL C01881 V=800.0 PL=0
MOVL C01882 V=800.0 PL=0
MOVL C01883 V=800.0 PL=0
MOVL C01884 V=800.0 PL=0
MOVL C01885 V=800.0 PL=0
MOVL C01886 V=800.0 PL=0
MOVL C01887 V=800.0 PL=0
MOVL C01888 V=800.0 PL=0
MOVL C01889 V=800.0 PL=0
MOVL C01890 V=800.0 PL=0
MOVL C01891 V=800.0 PL=0
MOVL C01892 V=800.0 PL=0
MOVL C01893 V=800.0 PL=0
MOVL C01894 V=800.0 PL=0
MOVL C01895 V=800.0 PL=0
MOVL C01896 V=800.0 PL=0
MOVL C01897 V=800.0 PL=0
MOVL C01898 V=800.0 PL=0
MOVL C01899 V=800.0 PL=0
MOVL C01900 V=800.0 PL=0
MOVL C01901 V=800.0 PL=0
MOVL C01902 V=800.0 PL=0
MOVL C01903 V=800.0 PL=0
MOVL C01904 V=800.0 PL=0
MOVL C01905 V=800.0 PL=0
MOVL C01906 V=800.0 PL=0
MOVL C01907 V=800.0 PL=0
MOVL C01908 V=800.0 PL=0
MOVL C01909 V=800.0 PL=0
MOVL C01910 V=800.0 PL=0
MOVL C01911 V=800.0 PL=0
MOVL C01912 V=800.0 PL=0
MOVL C01913 V=800.0 PL=0
MOVL C01914 V=800.0 PL=0
MOVL C01915 V=800.0 PL=0
MOVL C01916 V=800.0 PL=0
MOVL C01917 V=800.0 PL=0
MOVL C01918 V=800.0 PL=0
MOVL C01919 V=800.0 PL=0
MOVL C01920 V=800.0 PL=0
MOVL C01921 V=800.0 PL=0
MOVL C01922 V=800.0 PL=0
MOVL C01923 V=800.0 PL=0
MOVL C01924 V=800.0 PL=0
MOVL C01925 V=800.0 PL=0
MOVL C01926 V=800.0 PL=0
MOVL C01927 V=800.0 PL=0
MOVL C01928 V=800.0 PL=0
MOVL C01929 V=800.0 PL=0
MOVL C01930 V=800.0 PL=0
MOVL C01931 V=800.0 PL=0
MOVL C01932 V=800.0 PL=0
MOVL C01933 V=800.0 PL=0
MOVL C01934 V=800.0 PL=0
MOVL C01935 V=800.0 PL=0
MOVL C01936 V=800.0 PL=0
MOVL C01937 V=800.0 PL=0
MOVL C01938 V=800.0 PL=0
MOVL C01939 V=800.0 PL=0
MOVL C01940 V=800.0 PL=0
MOVL C01941 V=800.0 PL=0
MOVL C01942 V=800.0 PL=0
MOVL C01943 V=800.0 PL=0
MOVL C01944 V=800.0 PL=0
MOVL C01945 V=800.0 PL=0
MOVL C01946 V=800.0 PL=0
MOVL C01947 V=800.0 PL=0
MOVL C01948 V=800.0 PL=0
MOVL C01949 V=800.0 PL=0
MOVL C01950 V=800.0 PL=0
MOVL C01951 V=800.0 PL=0
MOVL C01952 V=800.0 PL=0
MOVL C01953 V=800.0 PL=0
MOVL C01954 V=800.0 PL=0
MOVL C01955 V=800.0 PL=0
MOVL C01956 V=800.0 PL=0
MOVL C01957 V=800.0 PL=0
MOVL C01958 V=800.0 PL=0
MOVL C01959 V=800.0 PL=0
MOVL C01960 V=800.0 PL=0
MOVL C01961 V=800.0 PL=0
MOVL C01962 V=800.0 PL=0
MOVL C01963 V=800.0 PL=0
MOVL C01964 V=800.0 PL=0
MOVL C01965 V=800.0 PL=0
MOVL C01966 V=800.0 PL=0
MOVL C01967 V=800.0 PL=0
MOVL C01968 V=800.0 PL=0
MOVL C01969 V=800.0 PL=0
MOVL C01970 V=800.0 PL=0
MOVL C01971 V=800.0 PL=0
MOVL C01972 V=800.0 PL=0
MOVL C01973 V=800.0 PL=0
MOVL C01974 V=800.0 PL=0
MOVL C01975 V=800.0 PL=0
MOVL C01976 V=800.0 PL=0
MOVL C01977 V=800.0 PL=0
MOVL C01978 V=800.0 PL=0
MOVL C01979 V=800.0 PL=0
MOVL C01980 V=800.0 PL=0
MOVL C01981 V=800.0 PL=0
MOVL C01982 V=800.0 PL=0
MOVL C01983 V=800.0 PL=0
MOVL C01984 V=800.0 PL=0
MOVL C01985 V=800.0 PL=0
MOVL C01986 V=800.0 PL=0
MOVL C01987 V=800.0 PL=0
MOVL C01988 V=800.0 PL=0
MOVL C01989 V=800.0 PL=0
MOVL C01990 V=800.0 PL=0
MOVL C01991 V=800.0 PL=0
MOVL C01992 V=800.0 PL=0
MOVL C01993 V=800.0 PL=0
MOVL C01994 V=800.0 PL=0
MOVL C01995 V=800.0 PL=0
MOVL C01996 V=800.0 PL=0
MOVL C01997 V=800.0 PL=0
MOVL C01998 V=800.0 PL=0
MOVL C01999 V=800.0 PL=0
MOVL C02000 V=800.0 PL=0
MOVL C02001 V=800.0 PL=0
MOVL C02002 V=800.0 PL=0
MOVL C02003 V=800.0 PL=0
MOVL C02004 V=800.0 PL=0
MOVL C02005 V=800.0 PL=0
MOVL C02006 V=800.0 PL=0
MOVL C02007 V=800.0 PL=0
MOVL C02008 V=800.0 PL=0
MOVL C02009 V=800.0 PL=0
MOVL C02010 V=800.0 PL=0
MOVL C02011 V=800.0 PL=0
MOVL C02012 V=800.0 PL=0
MOVL C02013 V=800.0 PL=0
MOVL C02014 V=800.0 PL=0
MOVL C02015 V=800.0 PL=0
MOVL C02016 V=800.0 PL=0
MOVL C02017 V=800.0 PL=0
MOVL C02018 V=800.0 PL=0
MOVL C02019 V=800.0 PL=0
MOVL C02020 V=800.0 PL=0
MOVL C02021 V=800.0 PL=0
MOVL C02022 V=800.0 PL=0
MOVL C02023 V=800.0 PL=0
MOVL C02024 V=800.0 PL=0
MOVL C02025 V=800.0 PL=0
MOVL C02026 V=800.0 PL=0
MOVL C02027 V=800.0 PL=0
MOVL C02028 V=800.0 PL=0
MOVL C02029 V=800.0 PL=0
MOVL C02030 V=800.0 PL=0
MOVL C02031 V=800.0 PL=0
MOVL C02032 V=800.0 PL=0
MOVL C02033 V=800.0 PL=0
MOVL C02034 V=800.0 PL=0
MOVL C02035 V=800.0 PL=0
MOVL C02036 V=800.0 PL=0
MOVL C02037 V=800.0 PL=0
MOVL C02038 V=800.0 PL=0
MOVL C02039 V=800.0 PL=0
MOVL C02040 V=800.0 PL=0
MOVL C02041 V=800.0 PL=0
MOVL C02042 V=800.0 PL=0
MOVL C02043 V=800.0 PL=0
MOVL C02044 V=800.0 PL=0
MOVL C02045 V=800.0 PL=0
MOVL C02046 V=800.0 PL=0
MOVL C02047 V=800.0 PL=0
MOVL C02048 V=800.0 PL=0
MOVL C02049 V=800.0 PL=0
MOVL C02050 V=800.0 PL=0
MOVL C02051 V=800.0 PL=0
MOVL C02052 V=800.0 PL=0
MOVL C02053 V=800.0 PL=0
MOVL C02054 V=800.0 PL=0
MOVL C02055 V=800.0 PL=0
MOVL C02056 V=800.0 PL=0
MOVL C02057 V=800.0 PL=0
MOVL C02058 V=800.0 PL=0
MOVL C02059 V=800.0 PL=0
MOVL C02060 V=800.0 PL=0
MOVL C02061 V=800.0 PL=0
MOVL C02062 V=800.0 PL=0
MOVL C02063 V=800.0 PL=0
MOVL C02064 V=800.0 PL=0
MOVL C02065 V=800.0 PL=0
MOVL C02066 V=800.0 PL=0
MOVL C02067 V=800.0 PL=0
MOVL C02068 V=800.0 PL=0
MOVL C02069 V=800.0 PL=0
MOVL C02070 V=800.0 PL=0
MOVL C02071 V=800.0 PL=0
MOVL C02072 V=800.0 PL=0
MOVL C02073 V=800.0 PL=0
MOVL C02074 V=800.0 PL=0
MOVL C02075 V=800.0 PL=0
MOVL C02076 V=800.0 PL=0
MOVL C02077 V=800.0 PL=0
MOVL C02078 V=800.0 PL=0
MOVL C02079 V=800.0 PL=0
MOVL C02080 V=800.0 PL=0
MOVL C02081 V=800.0 PL=0
MOVL C02082 V=800.0 PL=0
MOVL C02083 V=800.0 PL=0
MOVL C02084 V=800.0 PL=0
MOVL C02085 V=800.0 PL=0
MOVL C02086 V=800.0 PL=0
MOVL C02087 V=800.0 PL=0
MOVL C02088 V=800.0 PL=0
MOVL C02089 V=800.0 PL=0
MOVL C02090 V=800.0 PL=0
MOVL C02091 V=800.0 PL=0
MOVL C02092 V=800.0 PL=0
MOVL C02093 V=800.0 PL=0
MOVL C02094 V=800.0 PL=0
MOVL C02095 V=800.0 PL=0
MOVL C02096 V=800.0 PL=0
MOVL C02097 V=800.0 PL=0
MOVL C02098 V=800.0 PL=0
MOVL C02099 V=800.0 PL=0
MOVL C02100 V=800.0 PL=0
MOVL C02101 V=800.0 PL=0
MOVL C02102 V=800.0 PL=0
MOVL C02103 V=800.0 PL=0
MOVL C02104 V=800.0 PL=0
MOVL C02105 V=800.0 PL=0
MOVL C02106 V=800.0 PL=0
MOVL C02107 V=800.0 PL=0
MOVL C02108 V=800.0 PL=0
MOVL C02109 V=800.0 PL=0
MOVL C02110 V=800.0 PL=0
MOVL C02111 V=800.0 PL=0
